# B&R Automation Studio project NAEUL004C00R13L518F00 (part 73)

#### Act_OpsRun2.st
```iecst
(** 2019-04-16 **)
ACTION Act_OpsRun2:

	(*Unloader's Lifter Magazine Layout*)
	(*
		Direction: -->> Left To Right -->>

	                      +----------+
	                      |          |
	                      |          |
	     (Lif=PosCSlt) US3|          |
	               [Mag 3]|          |
	                      |          |
	     (Lif=PosBSlt) US2|          |
	               [Mag 2]|          |
	                      |          |
	     (Lif=PosASlt) US1|          |
	               [Mag 1]|          |
	                      | Unloader |
	                      +----------+

		Note: Program Action Called For Lifter As Shown Above
		      Setup Lifter Program Parameters Accordingly

	For 2 lane magconv
	-eGotoOpsStep, eGotoOpsStep1 will consider lane 1; eGotoOpsStep2,eGotoOpsStep3 consider lane 2
	i. Lifter move position D,E ; Load, Unload pos
	ii. Lifter 2 move position G,H ; Load, Unload pos
	*)

	//===================== third sequence  Lifter 2 ================================================
	IF eGotoOpsStep2 <> eOpsStep2 THEN
		CASE eGotoOpsStep2 OF
			//During unload check ops is standby step
			LiftMagLifterUnload:
				IF eOpsStep = LifMagULStepStandby OR eOpsStep = LifMagULStepMagCmp THEN
					eOpsStep2	:= eGotoOpsStep2;
				END_IF

			LiftMagConvIdle:
				IF eOpsStep2 = LiftMagLifterLoad THEN
					usiMag2Rdy := LifterLoadPos;
					eOpsStep2	:= eGotoOpsStep2;
				ELSIF eOpsStep2 = LiftMagConvOUT THEN
					usiMag2Rdy := LifterNA;
					eOpsStep2	:= eGotoOpsStep2;
				ELSIF eOpsStep2 = LiftMagConvIN THEN
					usiMag2Rdy := LifterMagInProgress;
					eOpsStep2	:= eGotoOpsStep2;
				ELSE
					eOpsStep2	:= eGotoOpsStep2;
				END_IF

			LiftMagConvOUT:
				IF eOpsStep2 = LiftMagLifterUnload THEN
					usiMag2Rdy := LifterUnloadPos;
					eOpsStep2	:= eGotoOpsStep2;
				END_IF

			ELSE
				eOpsStep2	:= eGotoOpsStep2;
		END_CASE
	END_IF

	IF eOpsStep2 = eGotoOpsStep2 THEN
		IF bPaused = FALSE THEN

			CASE eOpsStep2 OF
				LiftMagConvInit:
					sStepTxt1	:= 'Lifter Conveyor 2 Initialization';

					IF bMagSetFullExit2 AND p_bLinkDIOutMagConv2EntSen THEN
						eLifterConv2Act	:= MagConvActExitClpr;
					ELSE
						eLifterConv2Act	:=  MagConvActInitClpStop;
					END_IF

					IF (p_eLifterMagConv2Stat = MagConvActInitClpStop OR p_eLifterMagConv2Stat = MagConvActExitClpr) AND p_eLifterMagConvStatus = Done THEN
						eLifterConv2Act	:= MagConvActIdle;
						eGotoOpsStep2 	:= LifMagULStepInitLif;

					END_IF
					bPaused	:= p_bStop OR p_bStep;

				LifMagULStepInitLif:
					sStepTxt1	:= 'Lifter 2 Initialization';
					IF p_bDIOutShutterCloseRS = TRUE THEN
						eLifter2Act	:= LifterActFullHm;
					END_IF

					IF p_eLifter2Status = Done AND p_eLifter2Stat = LifterActFullHm THEN
						eLifter2Act	:= LifterActIdle;

						eGotoOpsStep2	:= LiftMagConvIdle;

					END_IF
					bPaused	:= p_bStop OR p_bStep;

				LiftMagConvIdle:
					bMagSetFullExit2 := FALSE;
					IF p_bMagConvLanePrep THEN
						IF p_bMagPresentSen2 THEN //limit sensor ON
							//idle,standby
						ELSIF usiMag2Rdy = LifterLoadRdyTrans AND p_bMagPresentSen2 = FALSE THEN //mag2rdy = 2,Lifter inposition (load) and InMagConv ExitSen present
							eGotoOpsStep2 := LiftMagConvIN;
						ELSIF usiMag2Rdy = LifterNA
							AND p_bMagPresentSen2 = FALSE
							AND eOpsStep2 <> LifMagULStepInitLif
							AND p_bOutShutterExtended
							AND p_bLinkDIOutMagConv2EntSen = FALSE
							THEN
							eGotoOpsStep2 :=  LiftMagLifterLoad;
						END_IF

						//Lane 2 prep, magazine2 full
						IF p_bMagConvLanePrep
							AND pa_bMagDis[2] = FALSE
							AND a_bMagAllwMagPresent[2] = TRUE
							AND a_tyMagAllwBffrStat[2].bBffrFull = TRUE
							AND p_bOutShutterExtended
							THEN
							eMagNxtLoad		:= MagNxtLoadInvalid;
							eGotoOpsStep2	:= LiftMagLifterUnload;
						END_IF
					END_IF

					bPaused	:= p_bStop OR p_bStep;

				LiftMagConvIN:
					sStepTxt1	:= 'Lifter 2 Conveyor Entering';
					eLifterConv2Act	:=  MagConvActEntClpStop;

					IF p_eLifterMagConv2Stat = MagConvActEntClpStop AND p_eLifterMagConv2Status = Done THEN
						eLifterConv2Act	:=  MagConvActIdle;
						bLocalMag2InPos := TRUE;
						eGotoOpsStep2 := LiftMagConvIdle;
					END_IF
					bPaused	:= p_bStop OR p_bStep;

				LiftMagConvOUT:
					IF usiMag2Rdy = LifterUnloadRdyTrans THEN //Out mag allow and in position (unload)
						sStepTxt1	:= 'Lifter 2 Conveyor Exiting';
						eLifterConv2Act	:=  MagConvActExitClpr;
						bMagSetFullExit2 := TRUE;
					END_IF

					IF p_eLifterMagConv2Stat = MagConvActExitClpr AND p_eLifterMagConv2Status = Done THEN
						eLifterConv2Act	:=  MagConvActIdle;
						eGotoOpsStep2 := LiftMagConvIdle;
						bMagSetFullExit2 := FALSE;
					END_IF
					bPaused	:= p_bStop OR p_bStep;

				LiftMagLifterLoad:
					sStepTxt1	:= 'Move To Loading Position';
					IF eOpsStep2 <> LifMagULStepInitLif AND bLift2Move = FALSE THEN //AND eOpsStep2 <> LifMagULStepLifMov THEN
						eLifter2Act := LifterActGoGPos; //G,H,; load ,unload
					END_IF

					IF (p_eLifter2Status = Done AND p_eLifter2Stat = LifterActGoGPos)THEN
						eLifter2Act := LifterActIdle;
						eGotoOpsStep2 := LiftMagConvIdle;
					END_IF
					bPaused	:= p_bStop OR p_bStep;

				LiftMagLifterUnload:
					sStepTxt1	:= 'Move To Unload Position';
					IF eOpsStep2 <> LifMagULStepInitLif  AND bLift2Move = FALSE
						AND p_eLifter2Stat <> LifterActGoBSltPos THEN//AND eOpsStep2 <> LifMagULStepLifMov  THEN
						eMagNxtLoad		:= MagNxtLoadInvalid;
						eLifter2Act 	:= LifterActGoHPos; //G,H,; load ,unload
					END_IF

					IF (p_eLifter2Status = Done AND p_eLifter2Stat = LifterActGoHPos)THEN
						eLifter2Act := LifterActIdle;
						eGotoOpsStep2	:= LiftMagConvOUT;
					END_IF
					bPaused	:= p_bStop OR p_bStep;

				LifMagULStepStandby:

			END_CASE
		END_IF
	END_IF
END_ACTION
```

#### Act_OpsInfo.st
```iecst
ACTION Act_OpsInfo:

	//Reset
	udiStatus1	:= 0;
	udiStatus2  := 0;
	//Magazine Not Present
	a_bMagAllwMagPresent[1]	:= p_bMagPresentSen1;
	a_bMagAllwMagPresent[2]	:= p_bMagPresentSen2;
	a_bMagAllwMagPresent[3]	:= p_bMagPresentSen3;

	FOR udi := 1 TO 3 DO
		IF pa_bMagDis[udi] = FALSE AND a_bMagAllwMagPresent[udi] = TRUE THEN
			EXIT;
		END_IF
	END_FOR

	IF udi = 4 THEN
		IF eOpsStep > LifMagULStepInitLif THEN
			udiStatus1	:= 10000;
		END_IF
	END_IF

	//Magazine Is Full
	a_tyMagAllwBffrStat[1]	:= p_tyBufferStat1;
	a_tyMagAllwBffrStat[2]	:= p_tyBufferStat2;
	a_tyMagAllwBffrStat[3]	:= p_tyBufferStat3;

	//Insert Good / Bad Magazine
	IF p_bConvInitDone = TRUE AND p_bConvHvBrd = TRUE THEN

		FOR udi := 1 TO 3 DO
			IF pa_bMagDis[udi] = FALSE AND pa_bMagRej[udi] = TRUE THEN
				EXIT;
			END_IF
		END_FOR

		IF udi < 4 THEN
			//Reject Mode
			IF p_bConvGdBrd = TRUE THEN
				//Good Board Exist
				FOR udi1 := 1 TO 3 DO
					IF pa_bMagDis[udi1] = FALSE AND a_bMagAllwMagPresent[udi1] = TRUE AND pa_bMagRej[udi1] = FALSE THEN
						EXIT;
					END_IF
				END_FOR

				IF udi1 = 4 THEN
					udiStatus1	:= 10004;
				END_IF

			ELSE
				//Bad Board Exist
				FOR udi1 := 1 TO 3 DO
					IF pa_bMagDis[udi1] = FALSE AND a_bMagAllwMagPresent[udi1] = TRUE AND pa_bMagRej[udi1] = TRUE THEN
						EXIT;
					END_IF
				END_FOR

				IF udi1 = 4 THEN
					udiStatus1	:= 10005;
				END_IF

			END_IF

		ELSE
			//Non-Reject Mode
			FOR udi1 := 1 TO 3 DO
				IF pa_bMagDis[udi1] = FALSE AND a_bMagAllwMagPresent[udi1] = TRUE THEN
					EXIT;
				END_IF
			END_FOR

			IF udi1 = 4 THEN
				udiStatus1	:= 10004;
			END_IF

		END_IF

	END_IF

	IF pa_bMagDis[1] = FALSE
		AND pa_bMagDis[2] = FALSE
		AND pa_bMagDis[3] = FALSE
		AND a_bMagAllwMagPresent[1] = TRUE
		AND a_bMagAllwMagPresent[2] = TRUE
		AND a_bMagAllwMagPresent[3] = TRUE
		AND udiStatus1	<> 10008
		THEN

		IF a_tyMagAllwBffrStat[1].bBffrFull
			AND a_tyMagAllwBffrStat[2].bBffrFull
			AND a_tyMagAllwBffrStat[3].bBffrFull
			THEN
			udiStatus1	:= 10008;
		END_IF
	END_IF

	IF pa_bMagDis[1] = FALSE
		AND pa_bMagDis[2] = FALSE
		AND pa_bMagDis[3] = TRUE
		AND a_bMagAllwMagPresent[1] = TRUE
		AND a_bMagAllwMagPresent[2] = TRUE
		AND udiStatus1	<> 10006
		AND udiStatus1	<> 10008
		THEN

		IF (p_tyBufferStat1.diTtlGdBrd + p_tyBufferStat1.diTtlBadBrd
			+ p_tyBufferStat2.diTtlGdBrd + p_tyBufferStat2.diTtlBadBrd >=
			p_tyBufferStat1.diTtlBrdCap + p_tyBufferStat2.diTtlBrdCap - 1)

			THEN
			udiStatus1	:= 10006;

		END_IF
	END_IF

	IF pa_bMagDis[1] = FALSE
			AND pa_bMagDis[2] = FALSE
			AND pa_bMagDis[3] = FALSE
			AND a_bMagAllwMagPresent[1] = TRUE
			AND a_bMagAllwMagPresent[2] = TRUE
			AND a_bMagAllwMagPresent[3] = TRUE
			AND udiStatus1	<> 10007
			AND udiStatus1	<> 10008
			THEN

			IF (p_tyBufferStat1.diTtlGdBrd + p_tyBufferStat1.diTtlBadBrd
			+ p_tyBufferStat2.diTtlGdBrd + p_tyBufferStat2.diTtlBadBrd
			+ p_tyBufferStat3.diTtlGdBrd + p_tyBufferStat3.diTtlBadBrd>=
			p_tyBufferStat1.diTtlBrdCap
			+ p_tyBufferStat2.diTtlBrdCap
			+ p_tyBufferStat3.diTtlBrdCap - 1)

				THEN
				udiStatus1	:= 10007;

			END_IF
	END_IF

	FOR udi := 1 TO 3 DO
		IF pa_bMagDis[udi] = FALSE AND a_bMagAllwMagPresent[udi] = TRUE AND a_tyMagAllwBffrStat[udi].bBffrFull = TRUE THEN
				udiStatus1	:= 10001 + (udi - 1);

			EXIT;
		END_IF
	END_FOR

END_ACTION
```

#### Act_OpsRst.st - Do Not Change!!!
```iecst
(** 2019-03-25 **)
ACTION Act_OpsRst:

	udiStatus1	:= 0;

	eLifterAct		:= LifterActIdle;
	eLifter2Act		:= LifterActIdle;
	eLifterConvAct		:= MagConvActIdle;
	eLifterConv2Act		:= MagConvActIdle;
	eBufferAct1		:= BufferActIdle;
	eBufferAct2		:= BufferActIdle;
	eBufferAct3		:= BufferActIdle;
	eUSSMEMAAct1	:= SMEMAActIdle;
	eUSSMEMAAct2	:= SMEMAActIdle;
	eUSSMEMAAct3	:= SMEMAActIdle;

	usiMag1Rdy 	:= LifterNA;
	usiMag2Rdy	:= LifterNA;
END_ACTION
```

### OpsPosAllwGo.typ - not listed in the package file held
```iecst
(*2018-12-11*)
(**)
(**)
(**)

TYPE
	ePosUSAllwGoStep :
		(
		ePosUSAllwGoStepNA,
		ePosUSAllwGoStepInit,
		ePosUSAllwGoStepStdBy,
		ePosUSAllwGoUSCheck
		);
	ePosDSAllwGoStep :
		(
		ePosDSAllwGoStepNA,
		ePosDSAllwGoStepInit,
		ePosDSAllwGoStepStdBy,
		ePosDSAllwGoDSCheck
		);
END_TYPE
```

### OpsPosAllwGo.var - not listed in the package file held
```iecst
VAR
	p_OpsUSPosAllwGoStep : UDINT;
	p_OpsDSPosAllwGoStep : UDINT;
	p_OpsDSPosAllwGo : UDINT;
	p_OpsUSPosAllwGo : UDINT;
END_VAR
```

### OpsInMagConv.typ - Do Not Change!!!
```iecst
(*2018-12-11*)
(**)
(*Sequence*)

TYPE
	eInMagConvStep :
		(
		InMagConvStepNA,
		InMagConvStepInit,
		InMagConvStepChk,
		InMagConvStepOpsEntMag,
		InMagConvStepOpsExtChkMagSize,
		InMagConvStepOpsExtMag,
		InMagConvStepOpsEntToMid
		);
END_TYPE
```

### OpsInMagConv.var - Change By Project
```iecst
(*2019-03-25*)
(**)
(*Action & State & Status*)
(**)
(*Alarm*)
VAR
	p_OpsInMagConvAlmData : UDINT;
END_VAR
(**)
(*Output*)
VAR
	p_OpsInMagConvAct : UDINT;
	p_OpsInMagConv2Act : UDINT;
	p_OpsInMagConvStepTxt : UDINT;
	p_OpsInMagConvStepTxt1 : UDINT;
	p_OpsInMagConvPaused : UDINT;
END_VAR
(**)
VAR
	p_OpsInMagConvStepEntMag : UDINT;
	p_OpsInMagConvStepEntToMid : UDINT;
	p_OpsInMagConvStepExtMag : UDINT;
	p_OpsInMagConvUSSOTAct : UDINT;
	p_OpsInMagConv2USSOTAct : UDINT;
	p_OpsInMagConv2StepEntMag : UDINT;
	p_OpsInMagConv2StepEntToMid : UDINT;
	p_OpsInMagConv2StepExtMag : UDINT;
END_VAR
```

### Program Logical/Operations/MultiMag_InOutMagazineConv/OpsInMagConv (IEC) - 1.00.0 - 

#### InputRef.var
```iecst
(*2019-04-16*)
(**)
(*General*)
VAR
	p_udiRstErr : REFERENCE TO UDINT;
	p_bEn : REFERENCE TO BOOL;
	p_bDis : REFERENCE TO BOOL;
	p_bRun : REFERENCE TO BOOL;
	p_bStop : REFERENCE TO BOOL;
	p_bStep : REFERENCE TO BOOL;
END_VAR
(**)
(*Configuration*)
VAR
	p_eInMagConvStat : REFERENCE TO eMagConvAction;
	p_eInMagConvStatus : REFERENCE TO eFBStatus;
	p_eInMagConv2Stat : REFERENCE TO eMagConvAction;
	p_eInMagConv2Status : REFERENCE TO eFBStatus;
END_VAR
(**)
VAR
	p_bStepOpsEntMag : REFERENCE TO BOOL;
	p_bStepOpsEntMidMag : REFERENCE TO BOOL;
	p_bStepOpsExtMag : REFERENCE TO BOOL;
	p_bStepOpsEntMag2 : REFERENCE TO BOOL;
	p_bStepOpsEntMidMag2 : REFERENCE TO BOOL;
	p_bStepOpsExtMag2 : REFERENCE TO BOOL;
END_VAR
(**)
VAR
	p_bMagSelMiniMag : REFERENCE TO BOOL;
END_VAR
(**)
VAR
	p_bInMagConvExtSen : REFERENCE TO BOOL;
	p_bMagHeightChkSen : REFERENCE TO BOOL;
	p_eLiftMagConvStatus : REFERENCE TO eFBStatus;
	p_eLiftMagConv2Status : REFERENCE TO eFBStatus;
END_VAR
(**)
(*AGV SOT*)
VAR
	p_eAGVMagStat : REFERENCE TO eAGVMagAction;
	p_eAGVMagStatus : REFERENCE TO eFBStatus;
	p_bAGVMagMcRunRdy : REFERENCE TO BOOL;
	p_eUSSOTStat : REFERENCE TO eSOTAction;
	p_eUSSOTStatus : REFERENCE TO eFBStatus;
	p_eUSSOTStat2 : REFERENCE TO eSOTAction;
	p_eUSSOTStatus2 : REFERENCE TO eFBStatus;
	p_bUSSOTTransporting : REFERENCE TO BOOL;
	p_bUSSOTTransporting2 : REFERENCE TO BOOL;
	p_bUSSOTConvStart : REFERENCE TO BOOL;
	p_bUSSOTConvStop : REFERENCE TO BOOL;
	p_bUSSOTUSRdy : REFERENCE TO BOOL;
END_VAR
(**)
VAR
	p_sProgNm : REFERENCE TO STRING[15];
	p_bNtSettingsLoadDone : REFERENCE TO BOOL;
	p_bCurtainSensorStat : REFERENCE TO BOOL;
END_VAR
```

#### InputRef_Link.var
```iecst
(*2018-12-11*)
(**)
(*External Data*)
VAR
	p_bLinkOpsLifMagULInitDone1 : REFERENCE TO BOOL;
	p_bLinkOpsLifMagULInitDone2 : REFERENCE TO BOOL;
	p_diLinkLifterActualPos : REFERENCE TO DINT;
	p_diLinkLifter2ActualPos : REFERENCE TO DINT;
	p_diLinkLifterTopPos : REFERENCE TO DINT;
	p_diLinkLifterTopPos2 : REFERENCE TO DINT;
	bLifterTopPos : BOOL;
	bLifterTopPos2 : BOOL;
	p_bLinkExtStprExtended : REFERENCE TO BOOL;
	p_bLinkExtStprRetracted : REFERENCE TO BOOL;
	p_bLinkExtStpr2Retracted : REFERENCE TO BOOL;
	p_bLinkInMagConvEntSen : REFERENCE TO BOOL;
	p_bLinkInMagConvExtSen : REFERENCE TO BOOL;
	p_bLinkInMagConvMidSen : REFERENCE TO BOOL;
	p_bLinkInMagConv2EntSen : REFERENCE TO BOOL;
	p_bLinkInMagConv2ExtSen : REFERENCE TO BOOL;
	p_bLinkInMagConv2MidSen : REFERENCE TO BOOL;
	p_bLinkUIMagRun : REFERENCE TO BOOL;
	p_bLinkOpsLifterMagStepEntMag : REFERENCE TO BOOL;
	p_bLinkOpsLifterMagStepExtMag : REFERENCE TO BOOL;
	p_bLinkOpsLifterMagStepEntMag2 : REFERENCE TO BOOL;
	p_bLinkOpsLifterMagStepExtMag2 : REFERENCE TO BOOL;
	p_eLinkMcParamMagExMode : REFERENCE TO eMcMagExchangeMode;
END_VAR
```

#### Local.var
```iecst
(*2019-04-16*)
(**)
(*Local Action, State & Status*)
VAR
	eStatus : eFBStatus := Idle;
	udiStatus : UDINT := 0;
	udiStatus1 : UDINT := 0;
END_VAR
(**)
(*Local Alarm*)
VAR
	tyAlmData : tyAlmDat;
	a_tyAlmText : ARRAY[10000..10099] OF tyAlmTxt := [(sAlmText:='Invalid Magazine Size.'),(sAlmText:='Top Magazine Conveyor Full.'),98((0))];
END_VAR
(**)
(*Local Output*)
VAR
	sStepTxt : STRING[80];
	sStepTxt1 : STRING[80];
	bPaused : BOOL;
	bStepEnterMag : BOOL := FALSE;
	bStepEntToMid : BOOL := FALSE;
	bStepExitMag : BOOL := FALSE;
	bStepEnterMag2 : BOOL := FALSE;
	bStepEntToMid2 : BOOL := FALSE;
	bStepExitMag2 : BOOL := FALSE;
END_VAR
(**)
VAR
	eInMagConvAct : eMagConvAction;
	eInMagConv2Act : eMagConvAction;
END_VAR
(**)
(*Local Input*)
VAR
	udiRstErr : UDINT := 0;
	bEn : BOOL := TRUE;
	bDis : BOOL := FALSE;
	bRun : BOOL;
	bStop : BOOL;
	bStep : BOOL;
END_VAR
(**)
VAR
	eInMagConvStat : eMagConvAction;
	eInMagConvStatus : eFBStatus;
	eInMagConv2Stat : eMagConvAction;
	eInMagConv2Status : eFBStatus;
	eUSSOTAct : eSOTAction;
	eUSSOTAct2 : eSOTAction;
END_VAR
(**)
VAR
	bStepOpsEntMag : BOOL := FALSE;
	bStepOpsEntMidMag : BOOL := FALSE;
	bStepOpsExtMag : BOOL := FALSE;
	bStepOpsEntMag2 : BOOL := FALSE;
	bStepOpsEntMidMag2 : BOOL := FALSE;
	bStepOpsExtMag2 : BOOL := FALSE;
END_VAR
(**)
VAR
	bMagSelMiniMag : BOOL := FALSE;
END_VAR
(**)
VAR
	bInMagConvExtSen : BOOL;
	bMagHeightChkSen : BOOL;
	bCurtainSensorStat : BOOL;
END_VAR
(**)
VAR
	sProgNm : STRING[15] := 'OpsInMagConv';
	bNtSettingsLoadDone : BOOL := TRUE;
END_VAR
(**)
(*Local*)
VAR
	bRstErr : BOOL;
	udiRstErrOld : UDINT;
	bInitialDone : BOOL;
	bInitDone : BOOL;
	eOpsStep : eInMagConvStep := InMagConvStepNA;
	eGotoStep : eInMagConvStep := InMagConvStepInit;
	eOpsStep1 : eInMagConvStep := InMagConvStepNA;
	eGotoStep1 : eInMagConvStep := InMagConvStepInit;
	bMnlLoad : BOOL;
	bMnlLoad2 : BOOL;
	bLiftConvMagExist : BOOL;
	bLiftConvMagExist2 : BOOL;
	bMagManEx : BOOL;
	bMagAutoEx : BOOL;
	udiModuleNum : UDINT := 6111;
END_VAR
```

#### Act_Alarm.st
```iecst
(** 2019-03-25 **)
ACTION Act_Alarm:

	//Error
	IF EDGEPOS(eStatus = Error) THEN

		tyAlmData.sProgNm		:= p_sProgNm;
		tyAlmData.udiCode		:= udiStatus;
		tyAlmData.eSeverity		:= AlmSeverityError;
		tyAlmData.udiRunTime	:= tyAlmData.udiRunTime + 1;
		tyAlmData.bAlm			:= TRUE;
		tyAlmData.udiModuleNum  := udiModuleNum;
		g_sOpsInMagConvProgNm		:= p_sProgNm;

		//Get Error Message
		IF tyAlmData.udiCode < 10000 OR tyAlmData.udiCode > 10099 THEN
			tyAlmData.sAlmMsg	:= 'Unknown';
			tyAlmData.sRcyMsg	:= 'Unknown';
		ELSE
			tyAlmData.sAlmMsg	:= a_tyAlmText[tyAlmData.udiCode].sAlmText;
			tyAlmData.sRcyMsg	:= a_tyAlmText[tyAlmData.udiCode].sRcyText;
		END_IF

	ELSIF bRstErr AND (tyAlmData.udiCode <> 0) THEN

		tyAlmData.udiCode		:= 0;
		tyAlmData.eSeverity		:= AlmSeverityNA;
		tyAlmData.sAlmMsg		:= '';
		tyAlmData.sRcyMsg		:= '';
		tyAlmData.bAlm			:= FALSE;
	END_IF

END_ACTION
```

#### Act_AlarmInfo.st
```iecst
(** 2019-01-14 **)
ACTION Act_AlarmInfo:

	//Info
	tyAlmData.sProgNm		:= p_sProgNm;
	tyAlmData.udiCode		:= udiStatus1;
	tyAlmData.eSeverity		:= AlmSeverityInfo;
	tyAlmData.udiRunTime	:= tyAlmData.udiRunTime + 1;

	//Get Info Message
	IF tyAlmData.udiCode < 10000 OR tyAlmData.udiCode > 10099 THEN
		tyAlmData.sAlmMsg	:= 'Unknown';
		tyAlmData.sRcyMsg	:= 'Unknown';
	ELSE
		tyAlmData.sAlmMsg	:= a_tyAlmText[tyAlmData.udiCode].sAlmText;
		tyAlmData.sRcyMsg	:= a_tyAlmText[tyAlmData.udiCode].sRcyText;
	END_IF

END_ACTION
```

#### Act_Background.st
```iecst
(** 2019-04-16 **)
ACTION Act_Background:

	//Reset bPaused
	IF EDGENEG(p_bStop OR p_bStep) THEN
		bPaused	:= FALSE;
	END_IF

	IF eStatus <> Error AND p_bRun = TRUE THEN
		IF (p_bEn = TRUE) AND (p_bDis = FALSE) THEN
			Act_OpsRun;
			Act_OpsInMagInfo;
		ELSE
			bPaused	:= p_bStop OR p_bStep;
		END_IF

		IF EDGEPOS(p_bEn = FALSE OR p_bDis = TRUE) THEN
			Act_OpsRst;
		END_IF

	ELSIF eStatus <> Error THEN
		sStepTxt	:= 'Stop';
		sStepTxt1	:= 'Stop';
	ELSE
		sStepTxt	:= 'Error';
		sStepTxt1	:= 'Error';
	END_IF

	//Reset
	IF EDGENEG(p_bRun) OR EDGEPOS(eStatus = Error) THEN
		Act_OpsInitial;
		Act_OpsRst;
	END_IF

	//Reset Error
	IF (eStatus = Error) AND bRstErr THEN
		eStatus		:= Idle;
		udiStatus	:= 0;
	END_IF

END_ACTION
```

#### Act_InitGlobal.st
```iecst
(** 2019-04-16 **)
ACTION Act_InitGlobal:

	(* Always Change If Project Change *)

	//Pass Data To Link
	p_bLinkOpsLifMagULInitDone1 ACCESS p_OpsLifMagULStepInitDone1;
	p_bLinkOpsLifMagULInitDone2 ACCESS p_OpsLifMagULStepInitDone2;
	p_diLinkLifterActualPos ACCESS p_LifterBtmActualPos;
	p_diLinkLifter2ActualPos ACCESS p_Lifter2ActualPos;
	p_diLinkLifterTopPos ACCESS p_McParamLifterTopPos;
	p_diLinkLifterTopPos2 ACCESS p_McParamLifterTopPos2;
	p_bLinkExtStprExtended ACCESS p_PneuNoSenTopExtStprExtended;
	p_bLinkExtStprRetracted ACCESS p_PneuNoSenTopExtStprRetracted;
	p_bLinkExtStpr2Retracted ACCESS p_PneuNoSenTopExtStpr2Retracted;
	p_bLinkInMagConvEntSen ACCESS p_DIInMagConvEntSen;
	p_bLinkInMagConvExtSen ACCESS p_DIInMagConvExtSen;
	p_bLinkInMagConvMidSen ACCESS p_DIInMagConvMidSen;
	p_bLinkInMagConv2EntSen ACCESS p_DIInMagConv2EntSen;
	p_bLinkInMagConv2ExtSen ACCESS p_DIInMagConv2ExtSen;
	p_bLinkInMagConv2MidSen ACCESS p_DIInMagConv2MidSen;
	//	p_bLinkUIMagRun ACCESS p_UIMagRun;
	p_bLinkOpsLifterMagStepEntMag ACCESS p_OpsLifMagULStepEntMag1;
	p_bLinkOpsLifterMagStepExtMag ACCESS p_OpsLifMagULStepExtMag1;
	p_bLinkOpsLifterMagStepEntMag2 ACCESS p_OpsLifMagULStepEntMag2;
	p_bLinkOpsLifterMagStepExtMag2 ACCESS p_OpsLifMagULStepExtMag2;
	p_eLinkMcParamMagExMode ACCESS p_McParamMagExMode;

	//Pass Data To Internal Use
	p_udiRstErr ACCESS p_RstErrReset;
//	p_bEn ACCESS p_OpsLifMagULStepInitDone1;
	p_bRun ACCESS p_OpsRun;
	p_bStop ACCESS p_OpsStop;
	p_bStep ACCESS p_OpsStep;

	p_eInMagConvStat ACCESS p_InMagConvStat;
	p_eInMagConvStatus ACCESS p_InMagConvStatus;
	p_eInMagConv2Stat ACCESS p_InMagConv2Stat;
	p_eInMagConv2Status ACCESS p_InMagConv2Status;

	p_bInMagConvExtSen ACCESS p_DIInMagConvExtSen;
//	p_bMagHeightChkSen ACCESS p_DIMagHeightChkSen;

	p_eLiftMagConvStatus ACCESS p_LifterMagConvStatus;
	p_eLiftMagConv2Status ACCESS p_LifterMagConv2Status;

	//AGV
	p_eAGVMagStat ACCESS p_AGVMag1Stat;
	p_eAGVMagStatus ACCESS p_AGVMag1Status;
	p_bAGVMagMcRunRdy ACCESS p_AGVMag1McRunRdy;
	//USSOT
	p_eUSSOTStat ACCESS p_USSOT1Stat;
	p_eUSSOTStatus ACCESS p_USSOT1Status;
	p_bUSSOTTransporting ACCESS p_USSOT1Transporting;
	p_bUSSOTConvStart ACCESS p_USSOT1ConvStart;
	p_bUSSOTConvStop ACCESS p_USSOT1ConvStop;
	p_bUSSOTUSRdy ACCESS p_USSOT1USRdy;
	p_eUSSOTStat2 ACCESS p_USSOT2Stat;
	p_eUSSOTStatus2 ACCESS p_USSOT2Status;
	p_bUSSOTTransporting2 ACCESS p_USSOT2Transporting;

	//	p_bMagSelMiniMag ACCESS p_MagRcpCurrRcpMiniMag;

//	p_sProgNm ACCESS p_NtParamOpsULDInMagProgNm;
	p_bNtSettingsLoadDone ACCESS p_StartupNtSettingsLoadDone;
//	p_bCurtainSensorStat ACCESS p_CurtainSensorStat;

	(* Always Change If Project Change *)

END_ACTION
```

#### Act_InitLocal.st
```iecst
(** 2019-04-16 **)
ACTION Act_InitLocal:

	//Input Reference Link To Local Variable
	p_udiRstErr ACCESS ADR(udiRstErr);
	p_bEn ACCESS ADR(bEn);
	p_bDis ACCESS ADR(bDis);
	p_bRun ACCESS ADR(bRun);
	p_bStop ACCESS ADR(bStop);
	p_bStep ACCESS ADR(bStep);

	p_eInMagConvStat ACCESS ADR(eInMagConvStat);
	p_eInMagConvStatus ACCESS ADR(eInMagConvStatus);
	p_eInMagConv2Stat ACCESS ADR(eInMagConv2Stat);
	p_eInMagConv2Status ACCESS ADR(eInMagConv2Status);

	p_bStepOpsEntMag ACCESS ADR(bStepOpsEntMag);
	p_bStepOpsEntMidMag ACCESS ADR(bStepOpsEntMidMag);
	p_bStepOpsExtMag ACCESS ADR(bStepOpsExtMag);
	p_bStepOpsEntMag2 ACCESS ADR(bStepOpsEntMag2);
	p_bStepOpsEntMidMag2 ACCESS ADR(bStepOpsEntMidMag2);
	p_bStepOpsExtMag2 ACCESS ADR(bStepOpsExtMag2);

	p_bMagSelMiniMag ACCESS ADR(bMagSelMiniMag);

	p_bMagHeightChkSen ACCESS ADR(bMagHeightChkSen);
	p_bInMagConvExtSen ACCESS ADR(bInMagConvExtSen);
	p_bCurtainSensorStat ACCESS ADR(bCurtainSensorStat);

	p_sProgNm ACCESS ADR(sProgNm);
	p_bNtSettingsLoadDone ACCESS ADR(bNtSettingsLoadDone);

END_ACTION
```

#### Act_Link.st
```iecst
(** 2018-12-11 **)
ACTION Act_Link:

	bLifterTopPos		:= (ABS(p_diLinkLifterActualPos - p_diLinkLifterTopPos))<500;
	bLifterTopPos2		:= (ABS(p_diLinkLifter2ActualPos - p_diLinkLifterTopPos2))<500;

//	p_bStepOpsEntMag	:= p_bLinkOpsLifMagULInitDone1 = TRUE AND (p_bLinkUIMagRun = TRUE OR (p_bLinkInMagConvExtSen = FALSE AND p_bLinkInMagConvMidSen = TRUE));
	p_bStepOpsEntMag	:= p_bLinkInMagConvExtSen = FALSE AND p_bLinkInMagConvMidSen = TRUE;
	p_bStepOpsExtMag	:= p_bLinkOpsLifMagULInitDone1 = TRUE AND bLifterTopPos = TRUE AND p_bLinkExtStprRetracted = TRUE AND p_bLinkInMagConvExtSen = TRUE AND p_bLinkOpsLifterMagStepEntMag = TRUE;
	p_bStepOpsEntMidMag	:= p_bLinkInMagConvEntSen AND p_bLinkInMagConvMidSen = FALSE;

	p_bStepOpsEntMag2	:= p_bLinkInMagConv2ExtSen = FALSE AND p_bLinkInMagConv2MidSen = TRUE;
	p_bStepOpsExtMag2	:= p_bLinkOpsLifMagULInitDone2 = TRUE AND bLifterTopPos2 = TRUE AND p_bLinkExtStpr2Retracted = TRUE AND p_bLinkInMagConv2ExtSen = TRUE AND p_bLinkOpsLifterMagStepEntMag2 = TRUE;
	p_bStepOpsEntMidMag2:= p_bLinkInMagConv2EntSen AND p_bLinkInMagConv2MidSen = FALSE;

	//LiftConv Out magazine
	IF p_bLinkOpsLifterMagStepExtMag THEN
		bLiftConvMagExist := FALSE;
	END_IF
	IF p_bLinkOpsLifterMagStepExtMag2 THEN
		bLiftConvMagExist2 := FALSE;
	END_IF

	//Mag Exchange Mode
	CASE p_eLinkMcParamMagExMode OF
		McSetMagXcAutoManMode:
			bMagManEx := TRUE;
			bMagAutoEx := TRUE;

		McSetMagXcAutoMode:
			bMagManEx := FALSE;
			bMagAutoEx := TRUE;

		McSetMagXcManMode:
			bMagManEx := TRUE;
			bMagAutoEx := FALSE;

	END_CASE
END_ACTION
```

#### Init.st
```iecst
(** 2019-03-25 **)
PROGRAM _INIT

	(* Always Change If Project Change *)

	//Pass Address To Global Address For External Use
	//Action, State & Status

	//Alarm
	p_OpsInMagConvAlmData		:= ADR(tyAlmData);

	//Output
	p_OpsInMagConvAct			:= ADR(eInMagConvAct);
	p_OpsInMagConv2Act			:= ADR(eInMagConv2Act);
	p_OpsInMagConvUSSOTAct		:= ADR(eUSSOTAct);
	p_OpsInMagConv2USSOTAct		:= ADR(eUSSOTAct2);
	p_OpsInMagConvStepTxt		:= ADR(sStepTxt);
	p_OpsInMagConvStepTxt1		:= ADR(sStepTxt1);
	p_OpsInMagConvPaused		:= ADR(bPaused);

	p_OpsInMagConvStepEntMag	:= ADR(bStepEnterMag);
	p_OpsInMagConvStepEntToMid	:= ADR(bStepEntToMid);
	p_OpsInMagConvStepExtMag	:= ADR(bStepExitMag);

	p_OpsInMagConv2StepEntMag	:= ADR(bStepEnterMag2);
	p_OpsInMagConv2StepEntToMid	:= ADR(bStepEntToMid2);
	p_OpsInMagConv2StepExtMag	:= ADR(bStepExitMag2);

	(* Always Change If Project Change *)

END_PROGRAM
```

#### Act_OpsInitial.st - Do Not Change!!!
```iecst
(** 2019-01-16 **)
ACTION Act_OpsInitial:

	eGotoStep	:= InMagConvStepInit;
	eOpsStep	:= InMagConvStepNA;
	eGotoStep1	:= InMagConvStepInit;
	eOpsStep1	:= InMagConvStepNA;

	bStepEnterMag	:= FALSE;
	bStepEntToMid 	:= FALSE;
	bStepExitMag	:= FALSE;
	bStepEnterMag2	:= FALSE;
	bStepEntToMid2	:= FALSE;
	bStepExitMag2	:= FALSE;

END_ACTION
```

#### Act_OpsInMagInfo.st
```iecst
(** 2019-04-16 **)
ACTION Act_OpsInMagInfo:

	IF p_bLinkInMagConvMidSen = TRUE AND p_bLinkInMagConvExtSen = TRUE AND p_bCurtainSensorStat = TRUE THEN
		udiStatus1		:= 10001;//Top magazine conveyor full.
	ELSE
		udiStatus1		:= 0;
	END_IF

END_ACTION
```

#### Act_OpsRun.st
```iecst
(** 2019-04-16 **)
ACTION Act_OpsRun:

	IF eGotoStep <> eOpsStep THEN

		CASE eGotoStep OF

			ELSE
				eOpsStep	:= eGotoStep;

		END_CASE

	END_IF

	IF eGotoStep = eOpsStep THEN

		IF bPaused = FALSE THEN

			CASE eOpsStep OF
				InMagConvStepNA:
					sStepTxt	:= 'NA';

					eGotoStep	:= InMagConvStepInit;

					//					bPaused		:= p_bStop OR p_bStep;

				InMagConvStepInit:
					sStepTxt			:= 'Initializing Magazine Conveyor';
					eInMagConvAct		:= MagConvActInit;

					IF (p_eInMagConvStatus = Done AND p_eInMagConvStat = MagConvActInit)
						THEN
						eInMagConvAct			:= MagConvActIdle;
						eGotoStep			:= InMagConvStepChk;
					END_IF

				InMagConvStepChk:
					sStepTxt	:= 'Checking Input Magazine Conveyor Condition';

					IF bMagAutoEx AND p_bLinkInMagConvMidSen = FALSE THEN
						eUSSOTAct	:= SOTActRun;
					ELSE
						eUSSOTAct	:= SOTActIdle;
					END_IF

					IF p_bStepOpsExtMag = TRUE AND bLiftConvMagExist = FALSE THEN
						eGotoStep	:= InMagConvStepOpsExtMag;
					ELSIF p_bStepOpsEntMag = TRUE THEN
						eGotoStep	:= InMagConvStepOpsEntMag;
					ELSIF p_bUSSOTTransporting= TRUE THEN 		//SOT Comm
						eGotoStep	:= InMagConvStepOpsEntToMid;
					ELSIF p_bStepOpsEntMidMag = TRUE THEN
						bMnlLoad	:= TRUE;
						eGotoStep	:= InMagConvStepOpsEntToMid;
					END_IF

					IF p_bStepOpsExtMag = FALSE AND p_bStepOpsEntMag = FALSE AND p_eLiftMagConvStatus <> Busy THEN
						bPaused		:= p_bStop OR p_bStep;
						IF bPaused THEN
							eUSSOTAct	:= SOTActIdle;
						END_IF
					END_IF

				InMagConvStepOpsEntMag:
					sStepTxt	:= 'Entering Magazine';

					eInMagConvAct		:= MagConvActInit;

					IF p_eInMagConvStatus = Done AND p_eInMagConvStat = MagConvActInit THEN
						eInMagConvAct	:= MagConvActIdle;
						eGotoStep		:= InMagConvStepChk;

						bPaused	:= p_bStop OR p_bStep;
					END_IF

				InMagConvStepOpsExtChkMagSize:
					sStepTxt	:= 'Checking Magazine Size';

					IF p_bMagSelMiniMag = TRUE THEN
						IF p_bMagHeightChkSen = TRUE AND p_bInMagConvExtSen = TRUE THEN
							eStatus		:= Error;
							udiStatus	:= 10000;		// Invalid Magazine Size
						ELSE
							eGotoStep	:= InMagConvStepOpsExtMag;
						END_IF
					ELSE
						eGotoStep	:= InMagConvStepOpsExtMag;
					END_IF

				InMagConvStepOpsExtMag:
					sStepTxt	:= 'Exiting Magazine';

					eInMagConvAct		:= MagConvActExit;

					IF p_eInMagConvStatus = Done AND p_eInMagConvStat = MagConvActExit THEN
						bLiftConvMagExist := TRUE;
						eInMagConvAct	:= MagConvActIdle;
						eGotoStep		:= InMagConvStepChk;

						bPaused	:= p_bStop OR p_bStep;
					END_IF

				InMagConvStepOpsEntToMid:
					sStepTxt	:= 'Entering Magazine To Middle';

					eInMagConvAct		:= MagConvActInit;

					IF p_eInMagConvStatus = Done AND p_eInMagConvStat = MagConvActInit AND
						(bMnlLoad OR (p_eUSSOTStatus = Done AND p_eUSSOTStat = SOTActRun)) THEN
						bMnlLoad		:= FALSE;
						eInMagConvAct	:= MagConvActIdle;
						eUSSOTAct		:= SOTActIdle;
						eGotoStep		:= InMagConvStepChk;

						bPaused	:= p_bStop OR p_bStep;
					END_IF

			END_CASE

		END_IF

	ELSE
		bPaused	:= p_bStop OR p_bStep;

	END_IF

	Act_OpsRun2;

	//Operation Step Status
	bStepEnterMag		:= eOpsStep = InMagConvStepOpsEntMag;
	bStepEntToMid		:= eOpsStep = InMagConvStepOpsEntToMid;
	bStepExitMag		:= eOpsStep = InMagConvStepOpsExtMag;

END_ACTION
```

#### Act_OpsRun2.st
```iecst
(** 2019-04-16 **)
ACTION Act_OpsRun2:
	//InMagConv Lane2
	//**********************second sequence - InMag2 ********************************************************
	IF eGotoStep1 <> eOpsStep1 THEN

		CASE eGotoStep1 OF

			ELSE
				eOpsStep1	:= eGotoStep1;

		END_CASE

	END_IF

	IF eGotoStep1 = eOpsStep1 THEN

		IF bPaused = FALSE THEN

			CASE eOpsStep1 OF
				InMagConvStepNA:
					sStepTxt1	:= 'NA';

					eGotoStep1	:= InMagConvStepInit;

//					bPaused		:= p_bStop OR p_bStep;

				InMagConvStepInit:
					sStepTxt1			:= 'Initializing Magazine Conveyor';
					eInMagConv2Act		:= MagConvActInit;

					IF (p_eInMagConv2Status = Done AND p_eInMagConv2Stat = MagConvActInit)
						THEN
						eInMagConv2Act			:= MagConvActIdle;
						eGotoStep1				:= InMagConvStepChk;
					END_IF

				InMagConvStepChk:
					sStepTxt1	:= 'Checking Input Magazine Conveyor Condition';

					IF bMagAutoEx AND p_bLinkInMagConv2MidSen = FALSE THEN
						eUSSOTAct2	:= SOTActRun;
					ELSE
						eUSSOTAct2	:= SOTActIdle;
					END_IF

					IF p_bStepOpsExtMag2 = TRUE AND bLiftConvMagExist2 = FALSE THEN
						eGotoStep1	:= InMagConvStepOpsExtMag;
					ELSIF p_bStepOpsEntMag2 = TRUE THEN
						eGotoStep1	:= InMagConvStepOpsEntMag;
					ELSIF  p_bUSSOTTransporting2= TRUE THEN		//SOT Comm
						eGotoStep1	:= InMagConvStepOpsEntToMid;
					ELSIF p_bStepOpsEntMidMag2 = TRUE THEN
						bMnlLoad2	:= TRUE;
						eGotoStep1	:= InMagConvStepOpsEntToMid;
					END_IF

					IF p_bStepOpsExtMag2 = FALSE AND p_bStepOpsEntMag2 = FALSE AND p_eLiftMagConv2Status <> Busy THEN
						bPaused		:= p_bStop OR p_bStep;
						IF bPaused THEN
							eUSSOTAct2	:= SOTActIdle;
						END_IF
					END_IF

				InMagConvStepOpsEntMag:
					sStepTxt1	:= 'Entering Magazine';

					eInMagConv2Act		:= MagConvActInit;

					IF p_eInMagConv2Status = Done AND p_eInMagConv2Stat = MagConvActInit THEN
						eInMagConv2Act	:= MagConvActIdle;
						eGotoStep1		:= InMagConvStepChk;

						bPaused	:= p_bStop OR p_bStep;
					END_IF

				InMagConvStepOpsExtChkMagSize:
					sStepTxt1	:= 'Checking Magazine Size';

					IF p_bMagSelMiniMag = TRUE THEN
						IF p_bMagHeightChkSen = TRUE AND p_bInMagConvExtSen = TRUE THEN
							eStatus		:= Error;
							udiStatus	:= 10000;		// Invalid Magazine Size
						ELSE
							eGotoStep1	:= InMagConvStepOpsExtMag;
						END_IF
					ELSE
						eGotoStep1	:= InMagConvStepOpsExtMag;
					END_IF

				InMagConvStepOpsExtMag:
					sStepTxt1	:= 'Exiting Magazine';

					eInMagConv2Act		:= MagConvActExit;

					IF p_eInMagConv2Status = Done AND p_eInMagConv2Stat = MagConvActExit THEN
						bLiftConvMagExist2 := TRUE;
						eInMagConv2Act	:= MagConvActIdle;
						eGotoStep1		:= InMagConvStepChk;

						bPaused	:= p_bStop OR p_bStep;
					END_IF

				InMagConvStepOpsEntToMid:
					sStepTxt1	:= 'Entering Magazine To Middle';

					eInMagConv2Act		:= MagConvActInit;

					IF p_eInMagConv2Status = Done AND p_eInMagConv2Stat = MagConvActInit AND
						(bMnlLoad2 OR  (p_eUSSOTStatus2 = Done AND p_eUSSOTStat2 = SOTActRun)) THEN
						bMnlLoad2		:= FALSE;
						eInMagConv2Act	:= MagConvActIdle;
						eUSSOTAct2		:= SOTActIdle;
						eGotoStep1		:= InMagConvStepChk;

						bPaused	:= p_bStop OR p_bStep;
					END_IF

			END_CASE

		END_IF

	ELSE
		bPaused	:= p_bStop OR p_bStep;
	END_IF

	//Operation Step Status
	bStepEnterMag2		:= eOpsStep1 = InMagConvStepOpsEntMag;
	bStepEntToMid2		:= eOpsStep1 = InMagConvStepOpsEntToMid;
	bStepExitMag2		:= eOpsStep1 = InMagConvStepOpsExtMag;

END_ACTION
```

#### Act_OpsRst.st - Do Not Change!!!
```iecst
(** 2019-03-25 **)
ACTION Act_OpsRst:

	eInMagConvAct	:= MagConvActIdle;
	eInMagConv2Act	:= MagConvActIdle;
	eUSSOTAct	:= SOTActIdle;
	eUSSOTAct2	:= SOTActIdle;
	bMnlLoad	:= FALSE;
	bMnlLoad2	:= FALSE;

END_ACTION
```

### OpsOutMagConv.typ - Do Not Change!!!
```iecst
(*2018-12-11*)
(**)
(*Sequence*)

TYPE
	eOutMagConvStep :
		(
		OutMagConvStepNA,
		OutMagConvStepInit,
		OutMagConvStepChk,
		OutMagConvStepEntMag,
		OutMagConvStepEntToMid,
		OutMagConvStepExitMag,
		OutMagConvStepWaitForRmvMag
		);
END_TYPE
```

### OpsOutMagConv.var - Change By Project
```iecst
(*2019-03-25*)
(**)
(*Action & State & Status*)
(**)
(*Alarm*)
VAR
	p_OpsOutMagConvAlmData : UDINT;
END_VAR
(**)
(*Output*)
VAR
	p_OpsOutMagConvAct : UDINT;
	p_OpsOutMagConv2Act : UDINT;
	p_OpsOutMagConvDSSOTAct : UDINT;
	p_OpsOutMagConv2DSSOTAct : UDINT;
	p_OpsOutMagConvStepTxt : UDINT;
	p_OpsOutMagConvStepTxt1 : UDINT;
	p_OpsOutMagConvPaused : UDINT;
END_VAR
(**)
VAR
	p_OpsOutMagConvStepInitDone : UDINT;
	p_OpsOutMagConvStepEntMag : UDINT;
	p_OpsOutMagConvStepEntMidMag : UDINT;
	p_OpsOutMagConvStepExtMag : UDINT;
	p_OpsOutMagConvStepWaitToRmvMag : UDINT;
	p_OpsOutMagConv2StepInitDone : UDINT;
	p_OpsOutMagConv2StepEntMag : UDINT;
	p_OpsOutMagConv2StepEntMidMag : UDINT;
	p_OpsOutMagConv2StepExtMag : UDINT;
	p_OpsOutMagConv2StepWaitToRmvMag : UDINT;
END_VAR
```

### Program Logical/Operations/MultiMag_InOutMagazineConv/OpsOutMagConv (IEC) - 1.00.0 - 

#### InputRef.var
```iecst
(*2019-04-16*)
(**)
(*General*)
VAR
	p_udiRstErr : REFERENCE TO UDINT;
	p_bEn : REFERENCE TO BOOL;
	p_bDis : REFERENCE TO BOOL;
	p_bRun : REFERENCE TO BOOL;
	p_bStop : REFERENCE TO BOOL;
	p_bStep : REFERENCE TO BOOL;
END_VAR
(**)
(*Configuration*)
VAR
	p_eOutMagConvStat : REFERENCE TO eMagConvAction;
	p_eOutMagConvStatus : REFERENCE TO eFBStatus;
	p_eOutMagConv2Stat : REFERENCE TO eMagConvAction;
	p_eOutMagConv2Status : REFERENCE TO eFBStatus;
END_VAR
(**)
VAR
	p_bStepEntMag : REFERENCE TO BOOL;
	p_bStepEntMag2 : REFERENCE TO BOOL;
	p_bEntSen : REFERENCE TO BOOL;
	p_bMidSen : REFERENCE TO BOOL;
	p_bExtSen : REFERENCE TO BOOL;
	p_bEntSen2 : REFERENCE TO BOOL;
	p_bMidSen2 : REFERENCE TO BOOL;
	p_bExtSen2 : REFERENCE TO BOOL;
	p_bExitSig : REFERENCE TO BOOL;
	p_bExitSig2 : REFERENCE TO BOOL;
	p_bOpsMnlUnloadMag : REFERENCE TO BOOL;
	p_bOpsMnlUnloadMag2 : REFERENCE TO BOOL;
END_VAR
(**)
(*AGV SOT*)
VAR
	p_eAGVMagStat : REFERENCE TO eAGVMagAction;
	p_eAGVMagStatus : REFERENCE TO eFBStatus;
	p_bAGVMagMcRunRdy : REFERENCE TO BOOL;
	p_eDSSOTStat : REFERENCE TO eSOTAction;
	p_eDSSOTStatus : REFERENCE TO eFBStatus;
	p_eDSSOTStat2 : REFERENCE TO eSOTAction;
	p_eDSSOTStatus2 : REFERENCE TO eFBStatus;
	p_bDSSOTTransporting : REFERENCE TO BOOL;
	p_bDSSOTTransporting2 : REFERENCE TO BOOL;
	p_bDSSOTConvStart : REFERENCE TO BOOL;
	p_bDSSOTConvStop : REFERENCE TO BOOL;
END_VAR
(**)
VAR
	p_sProgNm : REFERENCE TO STRING[15];
	p_bNtSettingsLoadDone : REFERENCE TO BOOL;
END_VAR
```

#### InputRef_Link.var
```iecst
(*2018-12-11*)
(**)
(*External Data*)
VAR
	p_bLinkOpsLifMagULInitDone1 : REFERENCE TO BOOL;
	p_bLinkOpsLifMagULInitDone2 : REFERENCE TO BOOL;
	p_diLinkLifterActualPos : REFERENCE TO DINT;
	p_diLinkLifterBtmPos : REFERENCE TO DINT;
	p_diLinkLifter2ActualPos : REFERENCE TO DINT;
	p_diLinkLifterBtmPos2 : REFERENCE TO DINT;
	bLifterBtmPos : BOOL;
	bLifterBtmPos2 : BOOL;
	p_tyLinkBffrStat : REFERENCE TO tyBffrStat;
	p_tyLinkBffr2Stat : REFERENCE TO tyBffrStat;
	p_bLinkLifterLmtSW : REFERENCE TO BOOL;
	p_bLinkLifter2LmtSW : REFERENCE TO BOOL;
	p_bLinkLiftExitMag : REFERENCE TO BOOL;
	p_bLinkLiftExitMag2 : REFERENCE TO BOOL;
	p_tyLinkDISetting : REFERENCE TO tyDigitalInputSettings;
	p_eLinkMcParamMagExMode : REFERENCE TO eMcMagExchangeMode;
END_VAR
```

#### Local.var
```iecst
(*2019-04-16*)
(**)
(*Local Action, State & Status*)
VAR
	eStatus : eFBStatus := Idle;
	udiStatus : UDINT := 0;
END_VAR
(**)
(*Local Alarm*)
VAR
	tyAlmData : tyAlmDat;
	a_tyAlmText : ARRAY[10000..10099] OF tyAlmTxt;
END_VAR
(**)
(*Local Output*)
VAR
	sStepTxt : STRING[80];
	sStepTxt1 : STRING[80];
	bPaused : BOOL;
	bStepInitDone : BOOL := FALSE;
	bStepEnterMag : BOOL := FALSE;
	bStepEnterMidMag : BOOL := FALSE;
	bStepExitMag : BOOL := FALSE;
	bStepWaitMagToRmvMnl : BOOL := FALSE;
	bStepInitDone2 : BOOL := FALSE;
	bStepEnterMag2 : BOOL := FALSE;
	bStepEnterMidMag2 : BOOL := FALSE;
	bStepExitMag2 : BOOL := FALSE;
	bStepWaitMagToRmvMnl2 : BOOL := FALSE;
END_VAR
(**)
VAR
	eOutMagConvAct : eMagConvAction;
	eOutMagConv2Act : eMagConvAction;
	eDSSOTAct : eSOTAction;
	eDSSOTAct2 : eSOTAction;
END_VAR
(**)
(*Local Input*)
VAR
	udiRstErr : UDINT := 0;
	bEn : BOOL := TRUE;
	bDis : BOOL := FALSE;
	bRun : BOOL;
	bStop : BOOL;
	bStep : BOOL;
END_VAR
(**)
VAR
	eOutMagConvStat : eMagConvAction;
	eOutMagConvStatus : eFBStatus;
	eOutMagConv2Stat : eMagConvAction;
	eOutMagConv2Status : eFBStatus;
END_VAR
(* *)
VAR
	bStepEntMag : BOOL := FALSE;
	bStepEntMag2 : BOOL := FALSE;
	bEntSen : BOOL := FALSE;
	bMidSen : BOOL := FALSE;
	bExtSen : BOOL := FALSE;
	bEntSen2 : BOOL := FALSE;
	bMidSen2 : BOOL := FALSE;
	bExtSen2 : BOOL := FALSE;
	bExitSig : BOOL := FALSE;
	bExitSig2 : BOOL := FALSE;
	bOpsMnlUnloadMag : BOOL := FALSE;
	fbMagToRmv : TON := (IN:=TRUE,PT:=T#1s);
	fbMagToRmv2 : TON := (IN:=TRUE,PT:=T#1s);
END_VAR
(**)
VAR
	sProgNm : STRING[15] := 'OpsAW';
	bNtSettingsLoadDone : BOOL := TRUE;
END_VAR
(**)
(*Local*)
VAR
	bRstErr : BOOL;
	udiRstErrOld : UDINT;
	bInitialDone : BOOL;
	bInitDone : BOOL;
	eOpsStep : eOutMagConvStep := OutMagConvStepNA;
	eGotoStep : eOutMagConvStep := OutMagConvStepInit;
	eOpsStep1 : eOutMagConvStep := OutMagConvStepNA;
	eGotoStep1 : eOutMagConvStep := OutMagConvStepInit;
	bMagManEx : BOOL;
	bMagAutoEx : BOOL;
	udiModuleNum : UDINT := 6131;
END_VAR
```

#### Act_Alarm.st
```iecst
(** 2019-03-25 **)
ACTION Act_Alarm:

	//Error
	IF EDGEPOS(eStatus = Error) THEN

		tyAlmData.sProgNm		:= p_sProgNm;
		tyAlmData.udiCode		:= udiStatus;
		tyAlmData.eSeverity		:= AlmSeverityError;
		tyAlmData.udiRunTime	:= tyAlmData.udiRunTime + 1;
		tyAlmData.bAlm			:= TRUE;
		tyAlmData.udiModuleNum  := udiModuleNum;
		g_sOpsOutMagConvProgNm		:= p_sProgNm;
		//Get Error Message
		IF tyAlmData.udiCode < 10000 OR tyAlmData.udiCode > 10099 THEN
			tyAlmData.sAlmMsg	:= 'Unknown';
			tyAlmData.sRcyMsg	:= 'Unknown';
		ELSE
			tyAlmData.sAlmMsg	:= a_tyAlmText[tyAlmData.udiCode].sAlmText;
			tyAlmData.sRcyMsg	:= a_tyAlmText[tyAlmData.udiCode].sRcyText;
		END_IF

	ELSIF bRstErr AND (tyAlmData.udiCode <> 0) THEN

		tyAlmData.udiCode		:= 0;
		tyAlmData.eSeverity		:= AlmSeverityNA;
		tyAlmData.sAlmMsg		:= '';
		tyAlmData.sRcyMsg		:= '';
		tyAlmData.bAlm			:= FALSE;
	END_IF

END_ACTION
```

#### Act_Background.st
```iecst
(** 2019-04-16 **)
ACTION Act_Background:

	//Reset bPaused
	IF EDGENEG(p_bStop OR p_bStep) THEN
		bPaused	:= FALSE;
	END_IF

	IF eStatus <> Error AND p_bRun = TRUE THEN
		IF (p_bEn = TRUE) AND (p_bDis = FALSE) THEN
			Act_OpsRun;
		ELSE
			bPaused	:= p_bStop OR p_bStep;
		END_IF

		IF EDGEPOS(p_bEn = FALSE OR p_bDis = TRUE) THEN
			Act_OpsRst;
		END_IF

	ELSIF eStatus <> Error THEN
		sStepTxt	:= 'Stop';
		sStepTxt1	:= 'Stop';
	ELSE
		sStepTxt	:= 'Error';
		sStepTxt1	:= 'Error';
	END_IF

	//Reset
	IF EDGENEG(p_bRun) OR EDGEPOS(eStatus = Error) THEN
		Act_OpsInitial;
		Act_OpsRst;
	END_IF

	//Reset Error
	IF (eStatus = Error) AND bRstErr THEN
		eStatus		:= Idle;
		udiStatus	:= 0;
	END_IF

END_ACTION
```

#### Act_InitGlobal.st
```iecst
(** 2019-04-16 **)
ACTION Act_InitGlobal:

	(* Always Change If Project Change *)

	//Pass Data To Link
	p_bLinkOpsLifMagULInitDone1 ACCESS p_OpsLifMagULStepInitDone1;
	p_bLinkOpsLifMagULInitDone2 ACCESS p_OpsLifMagULStepInitDone2;
	p_diLinkLifterActualPos ACCESS p_LifterBtmActualPos;
	p_diLinkLifterBtmPos ACCESS p_McParamLifterBtmPos;
	p_diLinkLifter2ActualPos ACCESS p_Lifter2ActualPos;
	p_diLinkLifterBtmPos2 ACCESS p_McParamLifterBtmPos2;
	p_tyLinkBffrStat ACCESS p_Buffer1BffrStat;
	p_tyLinkBffr2Stat ACCESS p_Buffer2BffrStat;
	p_bLinkLifterLmtSW ACCESS p_DILifterLmtSW;
	p_bLinkLifter2LmtSW ACCESS p_DILifter2LmtSW;
	p_bLinkLiftExitMag	ACCESS p_OpsLifMagULStepExtMag1;
	p_bLinkLiftExitMag2	ACCESS p_OpsLifMagULStepExtMag2;
	p_tyLinkDISetting ACCESS p_NtParamDISettings;
	p_eLinkMcParamMagExMode ACCESS p_McParamMagExMode;

	//Pass Data To Internal Use
	p_udiRstErr ACCESS p_RstErrReset;
//	p_bEn ACCESS p_OpsInitULDStepInitDone;
	p_bRun ACCESS p_OpsRun;
	p_bStop ACCESS p_OpsStop;
	p_bStep ACCESS p_OpsStep;

	p_eOutMagConvStat ACCESS p_OutMagConvStat;
	p_eOutMagConvStatus ACCESS p_OutMagConvStatus;
	p_eOutMagConv2Stat ACCESS p_OutMagConv2Stat;
	p_eOutMagConv2Status ACCESS p_OutMagConv2Status;

	p_bEntSen ACCESS p_DIOutMagConvEntSen;
	p_bMidSen ACCESS p_DIOutMagConvMidSen;
	p_bExtSen ACCESS p_DIOutMagConvExtSen;
	p_bEntSen2 ACCESS p_DIOutMagConv2EntSen;
	p_bMidSen2 ACCESS p_DIOutMagConv2MidSen;
	p_bExtSen2 ACCESS p_DIOutMagConv2ExtSen;

	//p_bExitSig ACCESS ADR(bExitSig);

	//AGV
	p_eAGVMagStat ACCESS p_AGVMag1Stat;
	p_eAGVMagStatus ACCESS p_AGVMag1Status;
	p_bAGVMagMcRunRdy ACCESS p_AGVMag1McRunRdy;
	//DSSOT
	p_eDSSOTStat ACCESS p_DSSOT1Stat;
	p_eDSSOTStatus ACCESS p_DSSOT1Status;
	p_eDSSOTStat2 ACCESS p_DSSOT2Stat;
	p_eDSSOTStatus2 ACCESS p_DSSOT2Status;
	p_bDSSOTTransporting ACCESS p_DSSOT1Transporting;
	p_bDSSOTTransporting2 ACCESS p_DSSOT2Transporting;
	p_bDSSOTConvStart ACCESS p_DSSOT1ConvStart;
	p_bDSSOTConvStop ACCESS p_DSSOT1ConvStop;

	p_bOpsMnlUnloadMag ACCESS p_UIOpsMnlUnloadMag;
	p_bOpsMnlUnloadMag2 ACCESS p_UIOpsMnlUnloadMag2;

//	p_sProgNm ACCESS p_NtParamOpsULDOutMagProgNm;
	p_bNtSettingsLoadDone ACCESS p_StartupNtSettingsLoadDone;

	(* Always Change If Project Change *)

END_ACTION
```

#### Act_InitLocal.st
```iecst
(** 2019-04-16 **)
ACTION Act_InitLocal:

	//Output Reference Link To Local Variable
	p_udiRstErr ACCESS ADR(udiRstErr);
	p_bEn ACCESS ADR(bEn);
	p_bDis ACCESS ADR(bDis);
	p_bRun ACCESS ADR(bRun);
	p_bStop ACCESS ADR(bStop);
	p_bStep ACCESS ADR(bStep);

	p_eOutMagConvStat ACCESS ADR(eOutMagConvStat);
	p_eOutMagConvStatus ACCESS ADR(eOutMagConvStatus);
	p_eOutMagConv2Stat ACCESS ADR(eOutMagConv2Stat);
	p_eOutMagConv2Status ACCESS ADR(eOutMagConv2Status);

	p_bStepEntMag ACCESS ADR(bStepEntMag);
	p_bStepEntMag2 ACCESS ADR(bStepEntMag2);
	p_bEntSen ACCESS ADR(bEntSen);
	p_bMidSen ACCESS ADR(bMidSen);
	p_bExtSen ACCESS ADR(bExtSen);
	p_bEntSen2 ACCESS ADR(bEntSen2);
	p_bMidSen2 ACCESS ADR(bMidSen2);
	p_bExtSen2 ACCESS ADR(bExtSen2);
	p_bExitSig ACCESS ADR(bExitSig);
	p_bExitSig2 ACCESS ADR(bExitSig2);
	p_bOpsMnlUnloadMag ACCESS ADR(bOpsMnlUnloadMag);

	p_sProgNm ACCESS ADR(sProgNm);
	p_bNtSettingsLoadDone ACCESS ADR(bNtSettingsLoadDone);

END_ACTION
```

#### Act_Link.st
```iecst
(** 2018-12-11 **)
ACTION Act_Link:

	bLifterBtmPos	:= (ABS(p_diLinkLifterActualPos - p_diLinkLifterBtmPos))<500;
	bLifterBtmPos2	:= (ABS(p_diLinkLifter2ActualPos - p_diLinkLifterBtmPos2))<500;

	p_bStepEntMag	:= p_bLinkOpsLifMagULInitDone1 = TRUE AND bLifterBtmPos = TRUE AND (p_tyLinkBffrStat.bBffrFull = TRUE AND p_bLinkLifterLmtSW = TRUE) AND p_bLinkLiftExitMag;
	p_bStepEntMag2	:= p_bLinkOpsLifMagULInitDone2 = TRUE AND bLifterBtmPos2 = TRUE AND (p_tyLinkBffr2Stat.bBffrFull = TRUE AND p_bLinkLifter2LmtSW = TRUE) AND p_bLinkLiftExitMag2;

	//Mag Exchange Mode
	CASE p_eLinkMcParamMagExMode OF
		McSetMagXcAutoManMode:
			bMagManEx := TRUE;
			bMagAutoEx := TRUE;

		McSetMagXcAutoMode:
			bMagManEx := FALSE;
			bMagAutoEx := TRUE;

		McSetMagXcManMode:
			bMagManEx := TRUE;
			bMagAutoEx := FALSE;
	END_CASE

END_ACTION
```

#### Init.st
```iecst
(** 2019-03-25 **)
PROGRAM _INIT

	(* Always Change If Project Change *)

	//Pass Address To Global Address For External Use
	//Action, State & Status

	//Alarm
	p_OpsOutMagConvAlmData		:= ADR(tyAlmData);

	//Output
	p_OpsOutMagConvAct			:= ADR(eOutMagConvAct);
	p_OpsOutMagConv2Act			:= ADR(eOutMagConv2Act);
	p_OpsOutMagConvDSSOTAct		:= ADR(eDSSOTAct);
	p_OpsOutMagConv2DSSOTAct	:= ADR(eDSSOTAct2);
	p_OpsOutMagConvStepTxt		:= ADR(sStepTxt);
	p_OpsOutMagConvStepTxt1		:= ADR(sStepTxt1);
	p_OpsOutMagConvPaused		:= ADR(bPaused);

	p_OpsOutMagConvStepInitDone		:= ADR(bStepInitDone);
	p_OpsOutMagConvStepEntMag		:= ADR(bStepEnterMag);
	p_OpsOutMagConvStepEntMidMag	:= ADR(bStepEnterMidMag);
	p_OpsOutMagConvStepExtMag		:= ADR(bStepExitMag);
	p_OpsOutMagConvStepWaitToRmvMag	:= ADR(bStepWaitMagToRmvMnl);

	p_OpsOutMagConv2StepInitDone	:= ADR(bStepInitDone2);
	p_OpsOutMagConv2StepEntMag		:= ADR(bStepEnterMag2);
	p_OpsOutMagConv2StepEntMidMag	:= ADR(bStepEnterMidMag2);
	p_OpsOutMagConv2StepExtMag		:= ADR(bStepExitMag2);
	p_OpsOutMagConv2StepWaitToRmvMag	:= ADR(bStepWaitMagToRmvMnl2);

	(* Always Change If Project Change *)

END_PROGRAM
```

#### Act_OpsInitial.st - Do Not Change!!!
```iecst
(** 2019-01-16 **)
ACTION Act_OpsInitial:

	eGotoStep	:= OutMagConvStepInit;
	eOpsStep	:= OutMagConvStepNA;
	eGotoStep1	:= OutMagConvStepInit;
	eOpsStep1	:= OutMagConvStepNA;

	bStepEnterMag		:= FALSE;
	bStepEnterMidMag 	:= FALSE;
	bStepExitMag		:= FALSE;
	bStepEnterMag2		:= FALSE;
	bStepEnterMidMag2 	:= FALSE;
	bStepExitMag2		:= FALSE;

END_ACTION
```

#### Act_OpsRun.st
```iecst
(** 2019-04-16 **)
ACTION Act_OpsRun:

	IF eGotoStep <> eOpsStep THEN

		CASE eGotoStep OF
			OutMagConvStepEntMag:
				IF bMagAutoEx AND p_bExtSen = FALSE THEN
					eDSSOTAct	:= SOTActIdle;
				END_IF

				IF p_bStepEntMag = TRUE THEN
					eOpsStep	:= eGotoStep;
				ELSIF p_bMidSen AND p_bExtSen = FALSE AND p_eOutMagConvStat = MagConvActIdle THEN
					eOpsStep	:= eGotoStep;
				ELSIF p_bMidSen = FALSE AND p_bExtSen THEN
					eGotoStep	:= OutMagConvStepChk;
				ELSIF p_bEntSen = FALSE AND p_bMidSen AND p_bExtSen THEN
					eGotoStep	:= OutMagConvStepEntToMid;
				END_IF

			OutMagConvStepEntToMid:
				IF bMagAutoEx AND p_bExtSen THEN
					eDSSOTAct	:= SOTActRun;
				ELSE
					eDSSOTAct	:= SOTActIdle;
				END_IF

				IF  p_bExtSen = FALSE THEN
					eGotoStep	:= OutMagConvStepChk;
				ELSIF p_bDSSOTTransporting = TRUE THEN
					eGotoStep	:= OutMagConvStepExitMag;
				ELSIF p_bEntSen AND p_bMidSen = FALSE AND p_bExtSen THEN
					eOpsStep	:= eGotoStep;
				ELSIF p_bStepEntMag = TRUE THEN
					eOpsStep	:= eGotoStep;
				ELSIF p_bOpsMnlUnloadMag AND p_bExtSen THEN
					eGotoStep	:= OutMagConvStepWaitForRmvMag;
				END_IF
			ELSE
				eOpsStep		:= eGotoStep;

		END_CASE

	END_IF

	IF eGotoStep = eOpsStep THEN

		IF bPaused = FALSE THEN

			CASE eOpsStep OF
				OutMagConvStepNA:
					sStepTxt	:= 'Output Magazine Conveyor Standby';

					eGotoStep	:= OutMagConvStepInit;

					bPaused		:= p_bStop OR p_bStep;

				OutMagConvStepInit:
					sStepTxt			:= 'Initializing Magazine Conveyor';
					eOutMagConvAct		:= MagConvActInit;

					IF (p_eOutMagConvStatus = Done AND p_eOutMagConvStat = MagConvActInit)
						THEN
						eOutMagConvAct			:= MagConvActIdle;
						eGotoStep				:= OutMagConvStepChk;
					END_IF

				OutMagConvStepChk:
					sStepTxt	:= 'Magazine Checking';
					IF p_tyLinkDISetting.diOutMagConvExtSen <> 0 AND p_bExtSen = FALSE THEN
						eGotoStep		:= OutMagConvStepEntMag;
					ELSIF p_tyLinkDISetting.diOutMagConvMidSen <> 0 AND p_bMidSen = FALSE THEN
						eGotoStep		:= OutMagConvStepEntToMid;
					ELSIF  p_tyLinkDISetting.diOutMagConvEntSen <> 0 AND p_bEntSen = FALSE AND
						p_tyLinkDISetting.diOutMagConvMidSen = 0 AND
						p_tyLinkDISetting.diOutMagConvMidSen = 0 THEN //when only 1 EntSen
						eGotoStep		:= OutMagConvStepEntMag;
					ELSIF (p_bExitSig OR p_bDSSOTTransporting) AND p_bExtSen THEN
						eGotoStep		:= OutMagConvStepExitMag;
					ELSIF p_bExtSen AND p_bMidSen AND p_bOpsMnlUnloadMag = FALSE THEN
						IF bMagAutoEx AND p_bExtSen THEN
							eDSSOTAct	:= SOTActRun;
						ELSE
							eDSSOTAct	:= SOTActIdle;
						END_IF
					ELSIF p_bOpsMnlUnloadMag AND p_bExtSen THEN
						eGotoStep	:= OutMagConvStepWaitForRmvMag;
					END_IF

					bPaused		:= p_bStop OR p_bStep;

				OutMagConvStepEntMag:
					sStepTxt	:= 'Entering Magazine'; //enter to end (extsen)

					eOutMagConvAct		:= MagConvActEnt;

					IF p_eOutMagConvStatus = Done AND p_eOutMagConvStat = MagConvActEnt THEN
						eOutMagConvAct	:= MagConvActIdle;
						eGotoStep		:= OutMagConvStepChk;

						bPaused	:= p_bStop OR p_bStep;
					END_IF

				OutMagConvStepEntToMid:
					sStepTxt	:= 'Entering To Middle Magazine Conveyor';

					eOutMagConvAct		:= MagConvActEnt;

					IF p_eOutMagConvStatus = Done AND p_eOutMagConvStat = MagConvActEnt THEN
						eOutMagConvAct	:= MagConvActIdle;
						eGotoStep		:= OutMagConvStepChk;

						bPaused	:= p_bStop OR p_bStep;
					END_IF

				OutMagConvStepExitMag:
					sStepTxt	:= 'Exiting Magazine';

					eOutMagConvAct		:= MagConvActExit;

					IF p_eOutMagConvStatus = Done AND p_eOutMagConvStat = MagConvActExit AND
						p_eDSSOTStatus = Done AND p_eDSSOTStat = SOTActRun THEN

						eOutMagConvAct		:= MagConvActIdle;
						eDSSOTAct			:= SOTActIdle;
						eGotoStep			:= OutMagConvStepChk;

						bPaused	:= p_bStop OR p_bStep;
					END_IF

				OutMagConvStepWaitForRmvMag:

					sStepTxt  := 'Waiting Magazine To Remove Manually';

					eDSSOTAct   := SOTActIdle;
					fbMagToRmv(IN:= (p_bExtSen = FALSE));

					IF p_bOpsMnlUnloadMag = FALSE OR fbMagToRmv.Q THEN
						fbMagToRmv (IN:= FALSE);
						eGotoStep		:= OutMagConvStepChk;
					END_IF

					bPaused			:= p_bStop OR p_bStep;
			END_CASE

		END_IF

	ELSE
		bPaused	:= p_bStop OR p_bStep;
	END_IF

	Act_OpsRun2;

	//Operation Step Status
	bStepInitDone		:= eOpsStep > OutMagConvStepInit;
	bStepEnterMag		:= eOpsStep = OutMagConvStepEntMag;
	bStepEnterMidMag	:= eOpsStep	= OutMagConvStepEntToMid;
	bStepExitMag		:= eOpsStep = OutMagConvStepExitMag;
	bStepWaitMagToRmvMnl:= eOpsStep = OutMagConvStepWaitForRmvMag;

END_ACTION
```

#### Act_OpsRun2.st
```iecst
(** 2019-04-16 **)
ACTION Act_OpsRun2:
	//OutMagConv Lane2
	//***************** sequence 2  ****************************************************************
	IF eGotoStep1 <> eOpsStep1 THEN

		CASE eGotoStep1 OF
			OutMagConvStepEntMag:
				IF bMagAutoEx AND p_bExtSen2 = FALSE THEN
					eDSSOTAct2	:= SOTActIdle;
				END_IF

				IF p_bStepEntMag2 = TRUE THEN
					eOpsStep1	:= eGotoStep1;
				ELSIF p_bMidSen2 AND p_bExtSen2 = FALSE AND p_eOutMagConv2Stat = MagConvActIdle THEN
					eOpsStep1	:= eGotoStep1;
				ELSIF p_bMidSen2 = FALSE AND p_bExtSen2 THEN
					eGotoStep1	:= OutMagConvStepChk;
				ELSIF p_bEntSen2 = FALSE AND p_bMidSen2 AND p_bExtSen2 THEN
					eGotoStep1	:= OutMagConvStepEntToMid;
				END_IF

			OutMagConvStepEntToMid:
				IF bMagAutoEx AND p_bExtSen2 THEN
					eDSSOTAct2	:= SOTActRun;
				ELSE
					eDSSOTAct2	:= SOTActIdle;
				END_IF

				IF  p_bExtSen2 = FALSE THEN
					eGotoStep1	:= OutMagConvStepChk;
				ELSIF p_bDSSOTTransporting2 = TRUE THEN
					eGotoStep1	:= OutMagConvStepExitMag;
				ELSIF p_bEntSen2 AND p_bMidSen2 = FALSE AND p_bExtSen2 THEN
					eOpsStep1	:= eGotoStep1;
				ELSIF p_bStepEntMag2 = TRUE THEN
					eOpsStep1	:= eGotoStep1;
				ELSIF p_bOpsMnlUnloadMag2 AND p_bExtSen2 THEN
					eGotoStep1	:= OutMagConvStepWaitForRmvMag;
				END_IF
			ELSE
				eOpsStep1		:= eGotoStep1;

		END_CASE

	END_IF

	IF eGotoStep1 = eOpsStep1 THEN

		IF bPaused = FALSE THEN

			CASE eOpsStep1 OF
				OutMagConvStepNA:
					sStepTxt1	:= 'Output Magazine Conveyor Standby';

					eGotoStep1	:= OutMagConvStepInit;

					bPaused		:= p_bStop OR p_bStep;

				OutMagConvStepInit:
					sStepTxt1			:= 'Initializing Magazine Conveyor';
					eOutMagConv2Act		:= MagConvActInit;

					IF (p_eOutMagConv2Status = Done AND p_eOutMagConv2Stat = MagConvActInit)
						THEN
						eOutMagConv2Act			:= MagConvActIdle;
						eGotoStep1				:= OutMagConvStepChk;
					END_IF

				OutMagConvStepChk:
					sStepTxt1	:= 'Magazine Checking';
					IF p_tyLinkDISetting.diOutMagConv2ExtSen <> 0 AND p_bExtSen2 = FALSE THEN
						eGotoStep1		:= OutMagConvStepEntMag;
					ELSIF p_tyLinkDISetting.diOutMagConv2MidSen <> 0 AND p_bMidSen2 = FALSE THEN
						eGotoStep1		:= OutMagConvStepEntToMid;
					ELSIF  p_tyLinkDISetting.diOutMagConv2EntSen <> 0 AND p_bEntSen2 = FALSE AND
						p_tyLinkDISetting.diOutMagConvMidSen = 0 AND
						p_tyLinkDISetting.diOutMagConvMidSen = 0 THEN //when only 1 EntSen
						eGotoStep1		:= OutMagConvStepEntMag;
					ELSIF (p_bExitSig2 OR p_bDSSOTTransporting2) AND p_bExtSen2 THEN
						eGotoStep1		:= OutMagConvStepExitMag;
					ELSIF p_bExtSen2 AND p_bMidSen2 AND p_bOpsMnlUnloadMag2 = FALSE THEN
						IF bMagAutoEx AND p_bExtSen2 THEN
							eDSSOTAct2	:= SOTActRun;
						ELSE
							eDSSOTAct2	:= SOTActIdle;
						END_IF
					ELSIF p_bOpsMnlUnloadMag2 AND p_bExtSen2 THEN
						eGotoStep1	:= OutMagConvStepWaitForRmvMag;
					END_IF

					bPaused		:= p_bStop OR p_bStep;

				OutMagConvStepEntMag:
					sStepTxt1	:= 'Entering Magazine'; //enter to end (extsen)

					eOutMagConv2Act		:= MagConvActEnt;

					IF p_eOutMagConv2Status = Done AND p_eOutMagConv2Stat = MagConvActEnt THEN
						eOutMagConv2Act	:= MagConvActIdle;
						eGotoStep1		:= OutMagConvStepChk;

						bPaused	:= p_bStop OR p_bStep;
					END_IF

				OutMagConvStepEntToMid:
					sStepTxt1	:= 'Entering To Middle Magazine Conveyor';

					eOutMagConv2Act		:= MagConvActEnt;

					IF p_eOutMagConv2Status = Done AND p_eOutMagConv2Stat = MagConvActEnt THEN
						eOutMagConv2Act	:= MagConvActIdle;
						eGotoStep1		:= OutMagConvStepChk;

						bPaused	:= p_bStop OR p_bStep;
					END_IF

				OutMagConvStepExitMag:
					sStepTxt1	:= 'Exiting Magazine';

					eOutMagConv2Act		:= MagConvActExit;

					IF p_eOutMagConv2Status = Done AND p_eOutMagConv2Stat = MagConvActExit AND
						p_eDSSOTStatus2 = Done AND p_eDSSOTStat2 = SOTActRun THEN

						eOutMagConv2Act		:= MagConvActIdle;
						eDSSOTAct2			:= SOTActIdle;
						eGotoStep1			:= OutMagConvStepChk;

						bPaused	:= p_bStop OR p_bStep;
					END_IF

				OutMagConvStepWaitForRmvMag:

					sStepTxt1  := 'Waiting Magazine To Remove Manually';

					eDSSOTAct2   := SOTActIdle;
					fbMagToRmv2(IN:= (p_bExtSen2 = FALSE));

					IF p_bOpsMnlUnloadMag2 = FALSE OR fbMagToRmv2.Q THEN
						fbMagToRmv2 (IN:= FALSE);
						eGotoStep1		:= OutMagConvStepChk;
					END_IF

					bPaused			:= p_bStop OR p_bStep;
			END_CASE

		END_IF

	ELSE
		bPaused	:= p_bStop OR p_bStep;
	END_IF

	//Operation Step Status
	bStepInitDone2		:= eOpsStep1 	> OutMagConvStepInit;
	bStepEnterMag2		:= eOpsStep1 	= OutMagConvStepEntMag;
	bStepEnterMidMag2	:= eOpsStep1	= OutMagConvStepEntToMid;
	bStepExitMag2		:= eOpsStep1	= OutMagConvStepExitMag;
	bStepWaitMagToRmvMnl2:= eOpsStep1 	= OutMagConvStepWaitForRmvMag;

END_ACTION
```

#### Act_OpsRst.st - Do Not Change!!!
```iecst
(** 2019-03-25 **)
ACTION Act_OpsRst:

	eOutMagConvAct	:= MagConvActIdle;
	eOutMagConv2Act	:= MagConvActIdle;
	eDSSOTAct	:= SOTActIdle;

END_ACTION
```

### OpsMagConvStpr.typ - Do Not Change!!!
```iecst
(*2018-12-11*)
(**)
(*Sequence*)

TYPE
	eMagConvStprRunStep :
		(
		MagConvStprStepNA,
		MagConvStprStepInit,
		MagConvStprStepChkCond,
		MagConvStprStepBtmLiftMagEnt,
		MagConvStprStepBtmLiftMagExit,
		MagConvStprStepTopLiftMagEnt,
		MagConvStprStepTopLiftMagExit,
		MagConvStprStepTopMagConvEnter,
		MagConvStprStepTopMagConvEnterD,
		MagConvStprStepBtmMagConvExit,
		MagConvStprStepDone,
		MagConvStprStepInitDone,
		MagConvStprStepBtmMagExitMnl
		);
END_TYPE
```

### OpsMagConvStpr.var - Change By Project
```iecst
(*2019-03-25*)
(**)
(*Action & State & Status*)
(**)
(*Alarm*)
VAR
	p_OpsMagConvStprAlmData : UDINT;
END_VAR
(**)
(*Output*)
VAR
	p_OpsMagConvStprStepTxt : UDINT;
	p_OpsMagConvStprPaused : UDINT;
	p_OpsMagConvStprBtmEntAct : UDINT;
	p_OpsMagConvStprBtmExitAct : UDINT;
	p_OpsMagConvStprBtmMidAct : UDINT;
	p_OpsMagConvStprTopEntAct : UDINT;
	p_OpsMagConvStprTopExitAct : UDINT;
	p_OpsMagConvStprTopMidAct : UDINT;
END_VAR
```

### Program Logical/Operations/MultiMag_InOutMagazineConv/OpsMagConvStpr (IEC) - 1.00.0 - 

#### Act_Alarm.st
```iecst
(** 2019-03-25 **)
ACTION Act_Alarm:

	//Error
	IF EDGEPOS(eStatus = Error) THEN

		tyAlmData.sProgNm		:= p_sProgNm;
		tyAlmData.udiCode		:= udiStatus;
		tyAlmData.eSeverity		:= AlmSeverityError;
		tyAlmData.udiRunTime	:= tyAlmData.udiRunTime + 1;
		tyAlmData.bAlm			:= TRUE;
		tyAlmData.udiModuleNum  := udiModuleNum;
		g_sOpsMagConvStprProgNm		:= p_sProgNm;
		//Get Error Message
		IF tyAlmData.udiCode < 10000 OR tyAlmData.udiCode > 10099 THEN
			tyAlmData.sAlmMsg	:= 'Unknown';
			tyAlmData.sRcyMsg	:= 'Unknown';
		ELSE
			tyAlmData.sAlmMsg	:= a_tyAlmText[tyAlmData.udiCode].sAlmText;
			tyAlmData.sRcyMsg	:= a_tyAlmText[tyAlmData.udiCode].sRcyText;
		END_IF

	ELSIF bRstErr AND (tyAlmData.udiCode <> 0) THEN

		tyAlmData.udiCode		:= 0;
		tyAlmData.eSeverity		:= AlmSeverityNA;
		tyAlmData.sAlmMsg		:= '';
		tyAlmData.sRcyMsg		:= '';

	END_IF

END_ACTION
```

#### Act_InitGlobal.st
```iecst
(** 2019-04-16 **)
ACTION Act_InitGlobal:

	(* Always Change If Project Change *)

	//Pass Data To Link
	p_bLinkOpsMnlUnloadMag ACCESS p_UIOpsMnlUnloadMag;
	p_bLinkOpsOutMagConvStepWaitRmv ACCESS p_OpsOutMagConvStepWaitToRmvMag;

	//Pass Data To Internal Use
	p_udiRstErr ACCESS p_RstErrReset;
	p_bRun ACCESS p_OpsRun;
	p_bStop ACCESS p_OpsStop;
	p_bStep ACCESS p_OpsStep;
	p_sProgNm ACCESS p_NtParamOpsMagConvStprProgNm;
	p_bNtSettingsLoadDone ACCESS p_StartupNtSettingsLoadDone;

	p_diLinkLiftBtmActualPos ACCESS p_LifterBtmActualPos;
	p_diLinkLiftBtmPos ACCESS p_McParamLifterBtmPos;
	p_diLinkLiftTopPos ACCESS p_McParamLifterTopPos;

	p_eStprBtmMidStat ACCESS p_PneuNoSenBtmMidStprStat;
	p_eStprBtmMidStatus ACCESS p_PneuNoSenBtmMidStprStatus;

	p_eStprBtmExitStat ACCESS p_PneuNoSenBtmExtStprStat;
	p_eStprBtmExitStatus ACCESS p_PneuNoSenBtmExtStprStatus;

	p_eStprTopEntStat ACCESS p_PneuNoSenTopEntStprStat;
	p_eStprTopEntStatus ACCESS p_PneuNoSenTopEntStprStatus;

	p_eStprTopMidStat ACCESS p_PneuNoSenTopMidStprStat;
	p_eStprTopMidStatus ACCESS p_PneuNoSenTopMidStprStatus;
	p_bStprTopMidStprExtended ACCESS p_PneuNoSenTopMidStprExtended;

	p_eStprTopExitStat ACCESS p_PneuNoSenTopExtStprStat;
	p_eStprTopExitStatus ACCESS p_PneuNoSenTopExtStprStatus;
	p_bStprTopExitStprExtended ACCESS p_PneuNoSenTopEntStprExtended;

	p_eInMagConvStatus ACCESS p_InMagConvStatus; 	//In magConv status
	p_eInMagConvStat ACCESS p_InMagConvStat; 	//In magConv status
	p_eOutMagConvStatus ACCESS p_OutMagConvStatus; 	//In magConv status
	p_eLiftMagConvStat ACCESS p_LifterMagConvStat; //LiftConv Status
	p_eLiftMagConvStatus ACCESS p_LifterMagConvStatus;

//	p_bBtmMagConvZ1Sen ACCESS p_DIBtmMagConvZ1Sen;
//	p_bTopMagConvZ1Sen ACCESS p_DITopMagConvZ1Sen;
	p_bBtmMagConvZ1Sen ACCESS p_DIOutMagConvEntSen;
	p_bTopMagConvZ1Sen ACCESS p_DIInMagConvExtSen;

	p_bBtmMagConvMidSen ACCESS p_DIOutMagConvMidSen; //LtoR view
	p_bTopMagConvMidSen ACCESS p_DIInMagConvMidSen;

	p_bBtmMagConvEndSen ACCESS p_DIOutMagConvExtSen; //LtoR view
	p_bTopMagConvEndSen ACCESS p_DIInMagConvEntSen;

	p_bMagPresentSen ACCESS p_DILifterLmtSW;

	p_bEnterSig ACCESS p_OpsInMagConvStepEntToMid;
	p_bExitSig ACCESS p_OpsOutMagConvStepExtMag;

	(* Always Change If Project Change *)

END_ACTION
```

#### Act_Link.st
```iecst
(** 2018-12-11 **)
ACTION Act_Link:

	IF (ABS(p_diLinkLiftBtmActualPos - p_diLinkLiftBtmPos))<500 THEN

		p_bLiftBtmPos	:= TRUE;

	ELSE
		p_bLiftBtmPos	:= FALSE;

	END_IF

	IF (ABS(p_diLinkLiftBtmActualPos - p_diLinkLiftTopPos))<500 THEN

		p_bLiftTopPos	:= TRUE;

	ELSE
		p_bLiftTopPos	:= FALSE;

	END_IF

	p_bBtmEntToLift		:= p_bMagPresentSen = FALSE AND p_bBtmMagConvZ1Sen AND ((p_eLiftMagConvStat = MagConvActEntStopClp (*OR p_eLiftMagConvStat = MagConvActInitStopClp*)) AND p_eLiftMagConvStatus = Busy) AND p_bLiftBtmPos;

	p_bTopExitFromLift	:= (p_eLiftMagConvStat = MagConvActExitClpr AND p_eLiftMagConvStatus = Busy) AND p_bLiftTopPos;

	p_bBtmExitFromLift	:=  (p_eLiftMagConvStat = MagConvActExitClpr AND p_eLiftMagConvStatus = Busy) AND p_bLiftBtmPos;

	p_bTopEntToLift		:= p_bMagPresentSen = FALSE AND p_bTopMagConvZ1Sen
							AND ((p_eLiftMagConvStat = MagConvActEntClpStop)
							AND p_eLiftMagConvStatus = Busy)
							AND p_bLiftTopPos;

	p_bTopEntFromMagConv := p_bEnterSig;// AND p_bTopMagConvEndSen;
	p_bBtmExitFromMagConv := p_bExitSig AND p_bBtmMagConvEndSen;
	p_bBtmExitMnl		 := p_bLinkOpsMnlUnloadMag AND p_bLinkOpsOutMagConvStepWaitRmv AND p_bBtmMagConvEndSen;

END_ACTION
```

#### Init.st
```iecst
(** 2019-03-25 **)
PROGRAM _INIT

	(* Always Change If Project Change *)

	//Pass Address To Global Address For External Use
	//Action, State & Status

	//Alarm
	p_OpsMagConvStprAlmData	:= ADR(tyAlmData);

	//Output
	p_OpsMagConvStprStepTxt		:= ADR(sStepTxt);
	p_OpsMagConvStprPaused		:= ADR(bPaused);
	p_OpsMagConvStprBtmEntAct	:= ADR(eStprBtmEntAct);
	p_OpsMagConvStprBtmExitAct	:= ADR(eStprBtmExitAct);
	p_OpsMagConvStprBtmMidAct   := ADR(eStprBtmMidAct);
	p_OpsMagConvStprTopEntAct	:= ADR(eStprTopEntAct);
	p_OpsMagConvStprTopExitAct	:= ADR(eStprTopExitAct);
	p_OpsMagConvStprTopMidAct	:= ADR(eStprTopMidAct);

	(* Always Change If Project Change *)

END_PROGRAM
```

#### Program Logical/Operations/MultiMag_InOutMagazineConv/OpsMagConvStpr/Sequence

##### Act_OpsRst.st
```iecst
(** 2019-03-25 **)
ACTION Act_OpsRst:

	eStprBtmExitAct	:= PneuActIdle;
	eStprBtmMidAct	:= PneuActIdle;
	eStprTopExitAct := PneuActIdle;
	eStprTopMidAct	:= PneuActIdle;

END_ACTION
```

### OpsMagConvStpr2.var - Change By Project
```iecst
(*2019-03-25*)
(**)
(*Action & State & Status*)
(**)
(*Alarm*)
VAR
	p_OpsMagConv2StprAlmData : UDINT;
END_VAR
(**)
(*Output*)
VAR
	p_OpsMagConv2StprStepTxt : UDINT;
	p_OpsMagConv2StprPaused : UDINT;
	p_OpsMagConv2StprBtmEntAct : UDINT;
	p_OpsMagConv2StprBtmExitAct : UDINT;
	p_OpsMagConv2StprBtmMidAct : UDINT;
	p_OpsMagConv2StprTopEntAct : UDINT;
	p_OpsMagConv2StprTopExitAct : UDINT;
	p_OpsMagConv2StprTopMidAct : UDINT;
END_VAR
```

### Program Logical/Operations/MultiMag_InOutMagazineConv/OpsMagConvStpr2 (IEC) - 1.00.0 - 

#### InputRef.var
```iecst
(*2019-04-16*)
(**)
(*General*)
VAR
	p_udiRstErr : REFERENCE TO UDINT;
	p_bEn : REFERENCE TO BOOL;
	p_bDis : REFERENCE TO BOOL;
	p_bRun : REFERENCE TO BOOL;
	p_bStop : REFERENCE TO BOOL;
	p_bStep : REFERENCE TO BOOL;
END_VAR
(**)
VAR
	p_bBtmEntToLift : REFERENCE TO BOOL;
	p_bBtmExitFromLift : REFERENCE TO BOOL;
	p_bTopEntToLift : REFERENCE TO BOOL;
	p_bTopExitFromLift : REFERENCE TO BOOL;
	p_bTopEntFromMagConv : REFERENCE TO BOOL;
	p_bBtmExitFromMagConv : REFERENCE TO BOOL;
	p_bBtmExitMnl : REFERENCE TO BOOL;
END_VAR
(**)
VAR
	p_eStprTopEntStat : REFERENCE TO ePneuAction;
	p_eStprTopEntStatus : REFERENCE TO eFBStatus;
END_VAR
(**)
VAR
	p_eStprBtmMidStat : REFERENCE TO ePneuAction;
	p_eStprBtmMidStatus : REFERENCE TO eFBStatus;
	p_eStprTopMidStat : REFERENCE TO ePneuAction;
	p_eStprTopMidStatus : REFERENCE TO eFBStatus;
	p_bStprTopMidStprExtended : REFERENCE TO BOOL;
END_VAR
(**)
VAR
	p_eStprBtmExitStat : REFERENCE TO ePneuAction;
	p_eStprBtmExitStatus : REFERENCE TO eFBStatus;
	p_eStprTopExitStat : REFERENCE TO ePneuAction;
	p_eStprTopExitStatus : REFERENCE TO eFBStatus;
	p_bStprTopExitStprExtended : REFERENCE TO BOOL;
END_VAR
(**)
VAR
	p_eLiftMagConvAct : REFERENCE TO eMagConvAction;
	p_eInMagConvStat : REFERENCE TO eMagConvAction;
	p_eInMagConvStatus : REFERENCE TO eFBStatus;
	p_eOutMagConvStatus : REFERENCE TO eFBStatus;
	p_eLiftMagConvStat : REFERENCE TO eMagConvAction;
	p_eLiftMagConvStatus : REFERENCE TO eFBStatus;
	p_bBtmMagConvZ1Sen : REFERENCE TO BOOL;
	p_bTopMagConvZ1Sen : REFERENCE TO BOOL;
	p_bTopMagConvMidSen : REFERENCE TO BOOL;
	p_bBtmMagConvMidSen : REFERENCE TO BOOL;
	p_bBtmMagConvEndSen : REFERENCE TO BOOL;
	p_bTopMagConvEndSen : REFERENCE TO BOOL;
	p_bMagPresentSen : REFERENCE TO BOOL;
END_VAR
(**)
VAR
	p_bLiftBtmPos : REFERENCE TO BOOL;
	p_bLiftTopPos : REFERENCE TO BOOL;
END_VAR
(**)
VAR
	p_bEnterSig : REFERENCE TO BOOL;
	p_bExitSig : REFERENCE TO BOOL;
END_VAR
(**)
VAR
	p_sProgNm : REFERENCE TO STRING[15];
	p_bNtSettingsLoadDone : REFERENCE TO BOOL;
END_VAR
```

#### InputRef_Link.var
```iecst
(*2018-12-11*)
(**)
VAR
	p_diLinkLiftBtmActualPos : REFERENCE TO DINT;
	p_diLinkLiftBtmPos : REFERENCE TO DINT;
	p_diLinkLiftTopPos : REFERENCE TO DINT;
	p_usiLinkProdRcpMcMode : REFERENCE TO USINT;
END_VAR
(**)
VAR
	p_bLinkOpsMnlUnloadMag : REFERENCE TO BOOL;
	p_bLinkOpsOutMagConvStepWaitRmv : REFERENCE TO BOOL;
END_VAR
```

#### Local.var
```iecst
(*2019-04-16*)
(**)
(*Local Action, State & Status*)
VAR
	eStatus : eFBStatus := Idle;
	udiStatus : UDINT := 0;
END_VAR
(**)
(*Local Alarm*)
VAR
	tyAlmData : tyAlmDat;
	a_tyAlmText : ARRAY[10000..10099] OF tyAlmTxt;
END_VAR
(**)
(*Local Output*)
VAR
	sStepTxt : STRING[80];
	bPaused : BOOL;
	eStprBtmEntAct : ePneuAction;
	eStprBtmMidAct : ePneuAction;
	eStprBtmExitAct : ePneuAction;
	eStprTopEntAct : ePneuAction;
	eStprTopMidAct : ePneuAction;
	eStprTopExitAct : ePneuAction;
	eLiftMagConvAct : ePneuAction;
END_VAR
(**)
(*Local Input*)
VAR
	udiRstErr : UDINT := 0;
	bEn : BOOL := TRUE;
	bDis : BOOL := FALSE;
	bRun : BOOL;
	bStop : BOOL;
	bStep : BOOL;
	eStprBtmMidStat : ePneuAction;
	eStprBtmMidStatus : eFBStatus;
	eStprBtmExitStatus : eFBStatus;
	eStprBtmExitStat : ePneuAction;
	eStprTopEntStat : ePneuAction;
	eStprTopEntStatus : eFBStatus;
	eStprTopMidStat : ePneuAction;
	eStprTopMidStatus : eFBStatus;
	eStprTopExitStat : ePneuAction;
	eStprTopExitStatus : eFBStatus;
	bLiftBtmPos : BOOL := FALSE;
	bLiftTopPos : BOOL;
	bBtmMagConvZ1Sen : BOOL;
	bTopMagConvZ1Sen : BOOL;
	bTopMagConvMidSen : BOOL;
	bBtmMagConvMidSen : BOOL;
	bBtmMagConvEndSen : BOOL;
	bTopMagConvEndSen : BOOL;
	bMagPresentSen : BOOL;
	sProgNm : STRING[15] := 'Ops1';
	bNtSettingsLoadDone : BOOL := TRUE;
	bBtmEntToLift : BOOL;
	bBtmExitFromLift : BOOL;
	bTopEntToLift : BOOL;
	bTopExitFromLift : BOOL;
	bTopEntFromMagConv : BOOL;
	bBtmExitFromMagConv : BOOL;
	bBtmExitMnl : BOOL;
	bEnterSig : BOOL;
	bExitSig : BOOL;
END_VAR
(**)
(*Local*)
VAR
	bRstErr : BOOL;
	udiRstErrOld : UDINT;
	bInitDone : BOOL;
	bInitialDone : BOOL;
	eOpsStep : eMagConvStprRunStep := MagConvStprStepNA;
	eGotoOpsStep : eMagConvStprRunStep := MagConvStprStepInit;
	eOpsStep1 : eMagConvStprRunStep := MagConvStprStepNA;
	eGotoOpsStep1 : eMagConvStprRunStep := MagConvStprStepInitDone;
	eOpsStep2 : eMagConvStprRunStep := MagConvStprStepNA;
	eGotoOpsStep2 : eMagConvStprRunStep := MagConvStprStepInit;
	fbMidChkDlyTm : TON := (PT:=T#1s);
	fbTopMidChkDlyTm : TON := (PT:=T#1s);
	udiModuleNum : UDINT;
END_VAR
```

#### Act_Alarm.st
```iecst
(** 2019-03-25 **)
ACTION Act_Alarm:

	//Error
	IF EDGEPOS(eStatus = Error) THEN

		tyAlmData.sProgNm		:= p_sProgNm;
		tyAlmData.udiCode		:= udiStatus;
		tyAlmData.eSeverity		:= AlmSeverityError;
		tyAlmData.udiRunTime	:= tyAlmData.udiRunTime + 1;
		tyAlmData.bAlm			:= TRUE;
		tyAlmData.udiModuleNum  := udiModuleNum;
		g_sOpsMagConvStpr2ProgNm		:= p_sProgNm;

		//Get Error Message
		IF tyAlmData.udiCode < 10000 OR tyAlmData.udiCode > 10099 THEN
			tyAlmData.sAlmMsg	:= 'Unknown';
			tyAlmData.sRcyMsg	:= 'Unknown';
		ELSE
			tyAlmData.sAlmMsg	:= a_tyAlmText[tyAlmData.udiCode].sAlmText;
			tyAlmData.sRcyMsg	:= a_tyAlmText[tyAlmData.udiCode].sRcyText;
		END_IF

	ELSIF bRstErr AND (tyAlmData.udiCode <> 0) THEN

		tyAlmData.udiCode		:= 0;
		tyAlmData.eSeverity		:= AlmSeverityNA;
		tyAlmData.sAlmMsg		:= '';
		tyAlmData.sRcyMsg		:= '';
		tyAlmData.bAlm			:= FALSE;
	END_IF

END_ACTION
```

#### Act_InitGlobal.st
```iecst
(** 2019-04-16 **)
ACTION Act_InitGlobal:

	(* Always Change If Project Change *)

	//Pass Data To Link
	p_bLinkOpsMnlUnloadMag ACCESS p_UIOpsMnlUnloadMag2;
	p_bLinkOpsOutMagConvStepWaitRmv ACCESS p_OpsOutMagConv2StepWaitToRmvMag;

	//Pass Data To Internal Use
	p_udiRstErr ACCESS p_RstErrReset;
	p_bRun ACCESS p_OpsRun;
	p_bStop ACCESS p_OpsStop;
	p_bStep ACCESS p_OpsStep;
//	p_sProgNm ACCESS p_NtParamOpsMagConv2StprProgNm;
	p_bNtSettingsLoadDone ACCESS p_StartupNtSettingsLoadDone;

	p_diLinkLiftBtmActualPos ACCESS p_Lifter2ActualPos;
	p_diLinkLiftBtmPos ACCESS p_McParamLifterBtmPos2;
	p_diLinkLiftTopPos ACCESS p_McParamLifterTopPos2;

	p_eStprBtmMidStat ACCESS p_PneuNoSenBtmMidStpr2Stat;
	p_eStprBtmMidStatus ACCESS p_PneuNoSenBtmMidStpr2Status;

	p_eStprBtmExitStat ACCESS p_PneuNoSenBtmExtStpr2Stat;
	p_eStprBtmExitStatus ACCESS p_PneuNoSenBtmExtStpr2Status;

	p_eStprTopEntStat ACCESS p_PneuNoSenTopEntStpr2Stat;
	p_eStprTopEntStatus ACCESS p_PneuNoSenTopEntStpr2Status;

	p_eStprTopMidStat ACCESS p_PneuNoSenTopMidStpr2Stat;
	p_eStprTopMidStatus ACCESS p_PneuNoSenTopMidStpr2Status;
	p_bStprTopMidStprExtended ACCESS p_PneuNoSenTopMidStpr2Extended;

	p_eStprTopExitStat ACCESS p_PneuNoSenTopExtStpr2Stat;
	p_eStprTopExitStatus ACCESS p_PneuNoSenTopExtStpr2Status;
	p_bStprTopExitStprExtended ACCESS p_PneuNoSenTopEntStpr2Extended;

	p_eInMagConvStatus ACCESS p_InMagConv2Status; 	//In magConv status
	p_eInMagConvStat ACCESS p_InMagConv2Stat; 		//In magConv status
	p_eOutMagConvStatus ACCESS p_OutMagConv2Status; //In magConv status
	p_eLiftMagConvStat ACCESS p_LifterMagConv2Stat; //LiftConv Status
	p_eLiftMagConvStatus ACCESS p_LifterMagConv2Status;

//	p_bBtmMagConvZ1Sen ACCESS p_DIBtmMagConvZ1Sen;
//	p_bTopMagConvZ1Sen ACCESS p_DITopMagConvZ1Sen;
	p_bBtmMagConvZ1Sen ACCESS p_DIOutMagConv2EntSen;
	p_bTopMagConvZ1Sen ACCESS p_DIInMagConv2ExtSen;

	p_bBtmMagConvMidSen ACCESS p_DIOutMagConv2MidSen; //LtoR view
	p_bTopMagConvMidSen ACCESS p_DIInMagConv2MidSen;

	p_bBtmMagConvEndSen ACCESS p_DIOutMagConv2ExtSen; //LtoR view
	p_bTopMagConvEndSen ACCESS p_DIInMagConv2EntSen;

	p_bMagPresentSen ACCESS p_DILifter2LmtSW;

	p_bEnterSig ACCESS p_OpsInMagConv2StepEntToMid;
	p_bExitSig ACCESS p_OpsOutMagConv2StepExtMag;

	(* Always Change If Project Change *)

END_ACTION
```

#### Act_InitLocal.st
```iecst
(** 2019-04-16 **)
ACTION Act_InitLocal:

	//Input Reference Link To Local Variable
	p_udiRstErr ACCESS ADR(udiRstErr);
	p_bEn ACCESS ADR(bEn);
	p_bDis ACCESS ADR(bDis);
	p_bRun ACCESS ADR(bRun);
	p_bStop ACCESS ADR(bStop);
	p_bStep ACCESS ADR(bStep);

	p_eStprBtmExitStat ACCESS ADR(eStprBtmExitStat);
	p_eStprBtmExitStatus ACCESS ADR(eStprBtmExitStatus);
	p_eStprBtmMidStat ACCESS ADR(eStprBtmMidStat);
	p_eStprBtmMidStatus ACCESS ADR(eStprBtmMidStatus);

	p_eStprTopExitStat ACCESS ADR(eStprTopExitStat);
	p_eStprTopExitStatus ACCESS ADR(eStprTopExitStatus);
	p_eStprTopMidStat ACCESS ADR(eStprTopMidStat);
	p_eStprTopMidStatus ACCESS ADR(eStprTopMidStatus);
	p_eStprTopEntStat ACCESS ADR(eStprTopEntStat);
	p_eStprTopEntStatus ACCESS ADR(eStprTopEntStatus);

	p_bLiftBtmPos ACCESS ADR(bLiftBtmPos);
	p_bLiftTopPos ACCESS ADR(bLiftTopPos);

	p_bBtmEntToLift ACCESS ADR(bBtmEntToLift);
	p_bBtmExitFromLift ACCESS ADR(bBtmExitFromLift);
	p_bTopEntToLift ACCESS ADR(bTopEntToLift);
	p_bTopExitFromLift ACCESS ADR(bTopExitFromLift);
	p_bBtmExitFromMagConv ACCESS ADR(bBtmExitFromMagConv);
	p_bTopEntFromMagConv ACCESS ADR(bTopEntFromMagConv);
	p_bBtmExitMnl ACCESS ADR(bBtmExitMnl);

	p_bBtmMagConvZ1Sen ACCESS ADR(bBtmMagConvZ1Sen);
	p_bTopMagConvZ1Sen ACCESS ADR(bTopMagConvZ1Sen);

	p_bTopMagConvMidSen ACCESS ADR(bTopMagConvMidSen);
	p_bBtmMagConvMidSen ACCESS ADR(bBtmMagConvMidSen);

	p_bBtmMagConvEndSen ACCESS ADR(bBtmMagConvEndSen);
	p_bTopMagConvEndSen ACCESS ADR(bTopMagConvEndSen);

	p_bMagPresentSen ACCESS ADR(bMagPresentSen);
	p_eLiftMagConvAct ACCESS ADR(eLiftMagConvAct);

	p_bEnterSig ACCESS ADR(bEnterSig);
	p_bExitSig ACCESS ADR(bExitSig);

	p_sProgNm ACCESS ADR(sProgNm);
	p_bNtSettingsLoadDone ACCESS ADR(bNtSettingsLoadDone);

END_ACTION
```

#### Init.st
```iecst
(** 2019-03-25 **)
PROGRAM _INIT

	(* Always Change If Project Change *)

	//Pass Address To Global Address For External Use
	//Action, State & Status

	//Alarm
	p_OpsMagConv2StprAlmData	:= ADR(tyAlmData);

	//Output
	p_OpsMagConv2StprStepTxt	:= ADR(sStepTxt);
	p_OpsMagConv2StprPaused		:= ADR(bPaused);
	p_OpsMagConv2StprBtmEntAct	:= ADR(eStprBtmEntAct);
	p_OpsMagConv2StprBtmExitAct	:= ADR(eStprBtmExitAct);
	p_OpsMagConv2StprBtmMidAct  := ADR(eStprBtmMidAct);
	p_OpsMagConv2StprTopEntAct	:= ADR(eStprTopEntAct);
	p_OpsMagConv2StprTopExitAct	:= ADR(eStprTopExitAct);
	p_OpsMagConv2StprTopMidAct	:= ADR(eStprTopMidAct);

	(* Always Change If Project Change *)

END_PROGRAM
```

#### Program Logical/Operations/MultiMag_InOutMagazineConv/OpsMagConvStpr2/Sequence

##### Act_OpsInitial.st
```iecst
(** 2019-01-16 **)
ACTION Act_OpsInitial:

	eOpsStep		:= MagConvStprStepNA;
	eGotoOpsStep	:= MagConvStprStepInit; //btm stpr
	eOpsStep1		:= MagConvStprStepNA;
	eGotoOpsStep1	:= MagConvStprStepInitDone; //top ent stpr
	eOpsStep2		:= MagConvStprStepNA;
	eGotoOpsStep2	:= MagConvStprStepInit; //top stpr

END_ACTION
```

##### Act_OpsRun.st
```iecst
(** 2019-04-16 **)
ACTION Act_OpsRun:

	IF eGotoOpsStep <> eOpsStep THEN

		CASE eGotoOpsStep OF

			ELSE
				eOpsStep	:= eGotoOpsStep;

		END_CASE

	END_IF

	IF eOpsStep = eGotoOpsStep THEN

		IF bPaused = FALSE THEN

			CASE eOpsStep OF

				MagConvStprStepInit:

					eStprBtmMidAct  := PneuActRet;
					eStprBtmExitAct	:= PneuActExt;

					IF (p_eStprBtmMidStat = PneuActRet AND p_eStprBtmMidStatus = Done) AND
						(p_eStprBtmExitStat = PneuActExt AND p_eStprBtmExitStatus = Done)
						THEN

						eStprBtmMidAct	:= PneuActIdle;
						eStprBtmExitAct	:= PneuActIdle;

						bPaused			:= p_bStop OR p_bStep;

						eGotoOpsStep	:= MagConvStprStepChkCond;

					END_IF

				MagConvStprStepChkCond:

					IF p_bBtmEntToLift THEN //opt
						eGotoOpsStep	:= MagConvStprStepBtmLiftMagEnt; //Bottom
					ELSIF p_bBtmExitFromLift THEN
						eGotoOpsStep	:= MagConvStprStepBtmLiftMagExit; //Bottom
					ELSIF p_bBtmExitFromMagConv THEN
						eGotoOpsStep    := MagConvStprStepBtmMagConvExit; //Bottom
					ELSIF p_bBtmExitMnl THEN
						eGotoOpsStep	:= MagConvStprStepBtmMagExitMnl; //Bottom
					ELSIF p_eLiftMagConvStatus = Done THEN
						eGotoOpsStep	:= MagConvStprStepDone;
					END_IF

					fbMidChkDlyTm (IN:=p_eOutMagConvStatus <> Busy);
					IF p_bBtmExitFromLift = FALSE AND p_bBtmEntToLift = FALSE AND p_bBtmExitFromMagConv = FALSE AND
						p_bBtmMagConvEndSen AND p_bBtmMagConvMidSen AND fbMidChkDlyTm.Q AND p_eInMagConvStatus <> Busy THEN
						eStprBtmMidAct  := PneuActExt;
					ELSIF fbMidChkDlyTm.Q THEN
						eStprBtmMidAct  := PneuActRet;
					END_IF

					IF ((p_eStprBtmMidStat = PneuActExt OR p_eStprBtmMidStat = PneuActRet) AND p_eStprBtmMidStatus = Done) THEN
						eStprBtmMidAct  := PneuActIdle;
						fbMidChkDlyTm (IN:=FALSE);
					END_IF

					bPaused	:= p_bStop OR p_bStep;

				MagConvStprStepBtmLiftMagEnt:

						eStprBtmMidAct  := PneuActExt;
						eStprBtmExitAct	:= PneuActRet;

					IF (p_eStprBtmMidStat = PneuActExt AND p_eStprBtmMidStatus = Done) AND
						(p_eStprBtmExitStat = PneuActRet AND p_eStprBtmExitStatus = Done) THEN

						eStprBtmMidAct  := PneuActIdle;
						eStprBtmExitAct	:= PneuActIdle;

						bPaused			:= p_bStop OR p_bStep;

						IF p_eLiftMagConvStatus = Done OR p_eLiftMagConvStatus = Idle THEN

							eGotoOpsStep	:= MagConvStprStepDone;

						END_IF

					END_IF

				MagConvStprStepBtmLiftMagExit:

					eStprBtmMidAct	:= PneuActRet;
					eStprBtmExitAct	:= PneuActExt;

					IF (p_eStprBtmMidStat = PneuActRet AND p_eStprBtmMidStatus = Done) AND
						(p_eStprBtmExitStat = PneuActExt AND p_eStprBtmExitStatus = Done) THEN

						eStprBtmMidAct   := PneuActIdle;
						eStprBtmExitAct	 := PneuActIdle;

						bPaused			:= p_bStop OR p_bStep;

						IF p_eLiftMagConvStatus = Done OR p_eLiftMagConvStatus = Idle THEN

							eGotoOpsStep	:= MagConvStprStepDone;

						END_IF
					END_IF

				MagConvStprStepBtmMagConvExit:
					eStprBtmMidAct	:= PneuActExt;
					eStprBtmExitAct	:= PneuActRet;
					IF (p_eStprBtmMidStat = PneuActExt AND p_eStprBtmMidStatus = Done) AND
						(p_eStprBtmExitStat = PneuActRet AND p_eStprBtmExitStatus = Done) THEN
						eStprBtmMidAct	:= PneuActIdle;
						eStprBtmExitAct	:= PneuActIdle;
						bPaused			:= p_bStop OR p_bStep;

						IF p_eOutMagConvStatus = Done OR p_eOutMagConvStatus = Idle THEN
							eGotoOpsStep	:= MagConvStprStepDone;
						END_IF
					END_IF

				MagConvStprStepDone:

					eStprBtmMidAct  := PneuActRet;
					eStprBtmExitAct	:= PneuActExt;

					IF (p_eStprBtmMidStat = PneuActRet AND p_eStprBtmMidStatus = Done) AND
						(p_eStprBtmExitStat = PneuActExt AND p_eStprBtmExitStatus = Done)
						THEN

						eStprBtmMidAct	:= PneuActIdle;
						eStprBtmExitAct	:= PneuActIdle;

						bPaused			:= p_bStop OR p_bStep;

						eGotoOpsStep	:= MagConvStprStepChkCond;

					END_IF
				MagConvStprStepInitDone:
					IF p_eInMagConvStatus = Done OR p_eInMagConvStatus = Idle THEN
						eStprTopEntAct  := PneuActExt;
					END_IF

					IF (p_eStprTopEntStat = PneuActExt AND p_eStprTopEntStatus = Done) THEN
						eStprTopEntAct  := PneuActIdle;
						eGotoOpsStep 	:= MagConvStprStepChkCond;
						bPaused			:= p_bStop OR p_bStep;
					END_IF

				MagConvStprStepBtmMagExitMnl:

					eStprBtmExitAct	:= PneuActRet;

					IF (p_eStprBtmExitStat = PneuActRet AND p_eStprBtmExitStatus = Done) THEN
						eStprBtmExitAct	 := PneuActIdle;

						IF p_bBtmExitMnl = FALSE THEN
							eGotoOpsStep	:= MagConvStprStepDone;
						END_IF

						bPaused			:= p_bStop OR p_bStep;
					END_IF

			END_CASE
		END_IF
	ELSE
		bPaused	:= p_bStop OR p_bStep;
	END_IF

	//==================== sequence 2 - Top entry stopper =============================================================
	IF eGotoOpsStep1 <> eOpsStep1 THEN
		CASE eGotoOpsStep1 OF
			ELSE
				eOpsStep1	:= eGotoOpsStep1;
		END_CASE
	END_IF

	IF eGotoOpsStep1 = eOpsStep1 THEN

		IF bPaused = FALSE THEN
			CASE eOpsStep1 OF
				MagConvStprStepInitDone:
					IF eOpsStep1 > MagConvStprStepInit THEN
						eStprTopEntAct  := PneuActExt;
					END_IF

					IF (p_eStprTopEntStat = PneuActExt AND p_eStprTopEntStatus = Done) THEN
						eStprTopEntAct  := PneuActIdle;
						eGotoOpsStep1 	:= MagConvStprStepChkCond;
						bPaused			:= p_bStop OR p_bStep;
					END_IF

				MagConvStprStepChkCond:
					IF p_bTopEntFromMagConv THEN
						eGotoOpsStep1    := MagConvStprStepTopMagConvEnter;
					END_IF
					bPaused	:= p_bStop OR p_bStep;

				MagConvStprStepTopMagConvEnter:
					eStprTopEntAct	:= PneuActRet;

					IF (p_eStprTopEntStat = PneuActRet AND p_eStprTopEntStatus = Done) THEN
						eStprTopEntAct   := PneuActIdle;
						eGotoOpsStep1	:= MagConvStprStepTopMagConvEnterD;
						bPaused			:= p_bStop OR p_bStep;

					END_IF
				MagConvStprStepTopMagConvEnterD:
					IF p_bTopMagConvMidSen OR (p_eInMagConvStatus <> Busy AND p_bTopMagConvEndSen =FALSE)THEN
						eStprTopEntAct	:= PneuActExt;
					END_IF

					IF (p_eStprTopEntStat = PneuActExt AND p_eStprTopEntStatus = Done) THEN
						eStprTopEntAct   := PneuActIdle;
						bPaused			:= p_bStop OR p_bStep;
						eGotoOpsStep1	:= MagConvStprStepChkCond;
					END_IF
			END_CASE
		END_IF
	ELSE
		bPaused	:= p_bStop OR p_bStep;
	END_IF

//################ sequence 3 - Top mid and ext stopper #####################################################################
	IF eGotoOpsStep2 <> eOpsStep2 THEN
		CASE eGotoOpsStep2 OF
			ELSE
				eOpsStep2	:= eGotoOpsStep2;
		END_CASE
	END_IF

	IF eGotoOpsStep2 = eOpsStep2 THEN
		IF bPaused = FALSE THEN
			CASE eOpsStep2 OF

				MagConvStprStepInit:

					eStprTopMidAct	:= PneuActRet;
					eStprTopExitAct := PneuActExt;

					IF 	(p_eStprTopMidStat = PneuActRet AND p_eStprTopMidStatus = Done) AND
						(p_eStprTopExitStat = PneuActExt AND p_eStprTopExitStatus = Done) THEN

						eStprTopMidAct	:= PneuActIdle;
						eStprTopExitAct := PneuActIdle;

						bPaused			:= p_bStop OR p_bStep;

						eGotoOpsStep2	:= MagConvStprStepChkCond;

					END_IF

				MagConvStprStepChkCond:

					IF p_bTopEntToLift THEN
						eGotoOpsStep2	:= MagConvStprStepTopLiftMagEnt;
					ELSIF p_bTopExitFromLift THEN //opt
						eGotoOpsStep2    := MagConvStprStepTopLiftMagExit;
					ELSIF p_eLiftMagConvStatus = Done THEN
						eGotoOpsStep2	:= MagConvStprStepDone;
					END_IF

					fbTopMidChkDlyTm (IN:=p_eInMagConvStatus <> Busy);
					IF p_bTopEntToLift = FALSE AND p_bTopExitFromLift = FALSE AND p_bTopEntFromMagConv = FALSE AND
						p_bTopMagConvZ1Sen AND p_bTopMagConvMidSen AND fbTopMidChkDlyTm.Q AND p_eOutMagConvStatus <> Busy THEN
						eStprTopMidAct  := PneuActExt;
					ELSIF fbTopMidChkDlyTm.Q THEN
						eStprTopMidAct  := PneuActRet;
					END_IF

					IF ((p_eStprTopMidStat = PneuActExt OR p_eStprTopMidStat = PneuActRet) AND p_eStprTopMidStatus = Done) THEN
						eStprTopMidAct  := PneuActIdle;
						fbTopMidChkDlyTm (IN:=FALSE);
					END_IF

					bPaused	:= p_bStop OR p_bStep;

				MagConvStprStepTopLiftMagEnt:
					IF p_bTopMagConvMidSen THEN
						eStprTopMidAct  := PneuActExt;
					ELSE
						eStprTopMidAct  := PneuActRet;
					END_IF
					eStprTopExitAct	:= PneuActRet;

					IF ((p_eStprTopMidStat = PneuActExt OR p_eStprTopMidStat = PneuActRet) AND p_eStprTopMidStatus = Done) AND
						(p_eStprTopExitStat = PneuActRet AND p_eStprTopExitStatus = Done) THEN

						eStprTopMidAct  := PneuActIdle;
						eStprTopExitAct	:= PneuActIdle;

						bPaused			:= p_bStop OR p_bStep;

						IF p_eLiftMagConvStatus = Done OR p_eLiftMagConvStatus = Idle THEN

							eGotoOpsStep2	:= MagConvStprStepDone;
						END_IF

					END_IF

				MagConvStprStepTopLiftMagExit:

					eStprTopMidAct	:= PneuActRet;
					eStprTopExitAct	:= PneuActRet;

					IF (p_eStprTopMidStat = PneuActRet AND p_eStprTopMidStatus = Done) AND
						(p_eStprTopExitStat = PneuActRet AND p_eStprTopExitStatus = Done) THEN

						eStprTopMidAct   := PneuActIdle;
						eStprTopExitAct	 := PneuActIdle;

						bPaused			:= p_bStop OR p_bStep;

						IF p_eLiftMagConvStatus = Done OR p_eLiftMagConvStatus = Idle THEN

							eGotoOpsStep2	:= MagConvStprStepDone;

						END_IF
					END_IF

				MagConvStprStepTopMagConvEnter:
					eStprTopEntAct	:= PneuActRet;

					IF (p_eStprTopEntStat = PneuActRet AND p_eStprTopEntStatus = Done) THEN
						eStprTopEntAct   := PneuActIdle;
						eGotoOpsStep2	:= MagConvStprStepTopMagConvEnterD;

						bPaused			:= p_bStop OR p_bStep;

					END_IF

				MagConvStprStepTopMagConvEnterD:
					IF p_bTopMagConvMidSen THEN
						eStprTopEntAct	:= PneuActExt;
					END_IF

					IF (p_eStprTopEntStat = PneuActExt AND p_eStprTopEntStatus = Done) THEN
						eStprTopEntAct   := PneuActIdle;
						bPaused			:= p_bStop OR p_bStep;
						eGotoOpsStep2	:= MagConvStprStepChkCond;
					END_IF

				MagConvStprStepDone:

					eStprTopMidAct	:= PneuActRet;
					eStprTopExitAct := PneuActExt;

					IF 	(p_eStprTopMidStat = PneuActRet AND p_eStprTopMidStatus = Done) AND
						(p_eStprTopExitStat = PneuActExt AND p_eStprTopExitStatus = Done) THEN

						eStprTopMidAct	:= PneuActIdle;
						eStprTopExitAct := PneuActIdle;

						bPaused			:= p_bStop OR p_bStep;

						eGotoOpsStep2	:= MagConvStprStepChkCond;

					END_IF

				MagConvStprStepInitDone:
					IF p_eInMagConvStatus = Done OR p_eInMagConvStatus = Idle THEN
						eStprTopEntAct  := PneuActExt;
					END_IF

					IF (p_eStprTopEntStat = PneuActExt AND p_eStprTopEntStatus = Done) THEN
						eStprTopEntAct  := PneuActIdle;
						eGotoOpsStep2 	:= MagConvStprStepChkCond;
						bPaused			:= p_bStop OR p_bStep;
					END_IF
			END_CASE
		END_IF
	ELSE
		bPaused	:= p_bStop OR p_bStep;
	END_IF

END_ACTION
```

### Program Logical/Operations/OpsPosAllwGo (IEC)

#### Init.st - Change By Project
```iecst
(** 2019-03-25 **)
PROGRAM _INIT
	p_OpsUSPosAllwGo	:= ADR(udiUSPosAllwGo);
	p_OpsDSPosAllwGo	:= ADR(udiDSPosAllwGo);
	p_OpsUSPosAllwGoStep	:= ADR(eOpsStep);
	p_OpsDSPosAllwGoStep	:= ADR(eOpsStep1);
END_PROGRAM
```

#### Act_InitGlobal.st - Change By Project
```iecst
(** 2019-04-16 **)
ACTION Act_InitGlobal:
	//Pass Data To Internal Use
	p_udiRstErr ACCESS p_RstErrReset;
	p_bRun ACCESS p_OpsRun;
	p_bStop ACCESS p_OpsStop;
	p_bStep ACCESS p_OpsStep;
	p_sProgNm ACCESS p_NtParamOpsMagConvStprProgNm;
	p_bNtSettingsLoadDone ACCESS p_StartupNtSettingsLoadDone;

	p_eUSCommMod1 ACCESS p_McParamUSCommAMod;
	p_eUSCommMod2 ACCESS p_McParamUSCommBMod;

	p_tyBufferStat1 ACCESS p_Buffer1BffrStat;
	p_tyBufferStat2 ACCESS p_Buffer2BffrStat;
	p_tyBufferStat3 ACCESS p_Buffer3BffrStat;

	p_dtBufferMagPresentTm1 ACCESS p_Buffer1MagPresentTm;
	p_dtBufferMagPresentTm2 ACCESS p_Buffer2MagPresentTm;
	p_dtBufferMagPresentTm3 ACCESS p_Buffer3MagPresentTm;

	p_bUSHermesUSRdy1 ACCESS p_USHermesAUSRdy;
	p_bUSHermesUSGdRdy1 ACCESS p_USHermesAUSGdRdy;

	p_bUSHermesUSRdy2 ACCESS p_USHermesBUSRdy;
	p_bUSHermesUSGdRdy2 ACCESS p_USHermesBUSGdRdy;

	p_bUSSMEMAUSRdy1 ACCESS p_USSMEMAAUSRdy;
	p_bUSSMEMAGdBrdRdy1 ACCESS p_USSMEMAAUSGdBrdRdy;
	p_bUSSMEMAUSRdy2 ACCESS p_USSMEMABUSRdy;
	p_bUSSMEMAGdBrdRdy2 ACCESS p_USSMEMABUSGdBrdRdy;

	p_bDSSMEMADSRdy1 ACCESS p_DSSMEMA1DSRdy;
	p_bDSSMEMADSRdy2 ACCESS p_DSSMEMA2DSRdy;
	p_bDSSMEMADSRdy3 ACCESS p_DSSMEMA3DSRdy;

	p_tyParamTravLif ACCESS p_OpsTravLifParamTravLif;
	p_bConvGdBrd ACCESS p_PshrConvGdBrd;

	p_usiLinkProdRcpCurrRcpMcMod ACCESS p_ProdRcpCurrRcp1McMod;

	p_bOpsModGoneThrough ACCESS p_OpsTravLifOpsModGonethrough;
END_ACTION
```

#### Act_Link.st - Change By Project
```iecst
(** 2018-12-11 **)
ACTION Act_Link:

	p_eULMod	:= USINT_TO_UDINT(p_usiLinkProdRcpCurrRcpMcMod);

	CASE p_eULMod OF
		ULModUnloadFrontLnA, ULModUnloadRearLnB, ULModUnloadDualLnAB:
			bBypsGdBadBrd	:= TRUE;
		ULModRejFrontLnA, ULModRejFrontLnARev, ULModRejRearLnB, ULModRejRearLnBRev, ULModRejDualLnA, ULModRejDualLnB:
			bBypsGdBadBrd	:= FALSE;
	END_CASE

	//Upstream
	IF p_eUSCommMod1 = McSetCommModHermes THEN
		bLocalUSRdy1	:= p_bUSHermesUSRdy1;
		bLocalUSGdRdy1	:= p_bUSHermesUSGdRdy1;
	ELSE
		bLocalUSRdy1	:= p_bUSSMEMAUSRdy1;
		bLocalUSGdRdy1	:= p_bUSSMEMAGdBrdRdy1;
	END_IF

	IF p_eUSCommMod2 = McSetCommModHermes THEN
		bLocalUSRdy2	:= p_bUSHermesUSRdy2;
		bLocalUSGdRdy2	:= p_bUSHermesUSGdRdy2;
	ELSE
		bLocalUSRdy2	:= p_bUSSMEMAUSRdy2;
		bLocalUSGdRdy2	:= p_bUSSMEMAGdBrdRdy2;
	END_IF

	IF p_eUSCommMod3 = McSetCommModHermes THEN
		bLocalUSRdy3	:= p_bUSHermesUSRdy3;
		bLocalUSGdRdy3	:= p_bUSHermesUSGdRdy3;
	ELSE
		bLocalUSRdy3	:= p_bUSSMEMAUSRdy3;
		bLocalUSGdRdy3	:= p_bUSSMEMAGdBrdRdy3;
	END_IF

	//Downstream
	IF p_eDSCommMod1 = McSetCommModHermes THEN
		bLocalDSRdy1	:= p_bDSHermesDSRdy1;
	ELSE
		bLocalDSRdy1	:= p_bDSSMEMADSRdy1;
	END_IF

	IF p_eDSCommMod2 = McSetCommModHermes THEN
		bLocalDSRdy2	:= p_bDSHermesDSRdy2;
	ELSE
		bLocalDSRdy2	:= p_bDSSMEMADSRdy2;
	END_IF

	IF p_eDSCommMod3 = McSetCommModHermes THEN
		bLocalDSRdy3	:= p_bDSHermesDSRdy3;
	ELSE
		bLocalDSRdy3	:= p_bDSSMEMADSRdy3;
	END_IF

END_ACTION
```

#### Act_InitLocal.st - Do Not Change!!!
```iecst
(** 2019-04-16 **)
ACTION Act_InitLocal:

	//Input Reference Link To Local Variable
	p_udiRstErr ACCESS ADR(udiRstErr);
	p_bEn ACCESS ADR(bEn);
	p_bDis ACCESS ADR(bDis);
	p_bRun ACCESS ADR(bRun);
	p_bStop ACCESS ADR(bStop);
	p_bStep ACCESS ADR(bStep);

	p_eUSCommMod1 ACCESS ADR(eUSCommMod1);
	p_eUSCommMod2 ACCESS ADR(eUSCommMod2);
	p_eUSCommMod3 ACCESS ADR(eUSCommMod3);
	p_eDSCommMod1 ACCESS ADR(eDSCommMod1);
	p_eDSCommMod2 ACCESS ADR(eDSCommMod2);
	p_eDSCommMod3 ACCESS ADR(eDSCommMod3);

	p_bUSSMEMAUSRdy3 ACCESS ADR(bUSSMEMAUSRdy3);
	p_bUSSMEMAGdBrdRdy3 ACCESS ADR(bUSSMEMAGdBrdRdy3);

	p_bDSHermesDSRdy1 ACCESS ADR(bDSHermesDSRdy1);
	p_bDSHermesDSRdy2 ACCESS ADR(bDSHermesDSRdy2);
	p_bDSHermesDSRdy3 ACCESS ADR(bDSHermesDSRdy3);

	p_sProgNm ACCESS ADR(sProgNm);
	p_bNtSettingsLoadDone ACCESS ADR(bNtSettingsLoadDone);

	p_bBypsGdBadBrd ACCESS ADR(bBypsGdBadBrd);
	p_eULMod ACCESS ADR(eULMode);

END_ACTION
```

#### Package Logical/Operations/OpsPosAllwGo/Sequence - Do Not Change!!!

#### Act_OpsInitial.st
```iecst
(** 2019-01-16 **)
ACTION Act_OpsInitial:

	eOpsStep		:= ePosUSAllwGoStepNA;
	eGotoOpsStep	:= ePosUSAllwGoStepInit;

	eOpsStep1		:= ePosDSAllwGoStepNA;
	eGotoOpsStep1	:= ePosDSAllwGoStepInit;
END_ACTION
```

#### Act_OpsRst.st
```iecst
(** 2019-03-25 **)
ACTION Act_OpsRst:

	udiUSPosAllwGo := 99;
	udiDSPosAllwGo := 99;

END_ACTION
```

#### Act_OpsRun.st
```iecst
(** 2019-04-16 **)
ACTION Act_OpsRun:
	bPaused	:= p_bStop OR p_bStep;

	IF eGotoOpsStep <> eOpsStep THEN

		CASE eGotoOpsStep OF

			ELSE
				eOpsStep	:= eGotoOpsStep;

		END_CASE

	END_IF

	IF eOpsStep = eGotoOpsStep THEN

		IF bPaused = FALSE THEN

			CASE eOpsStep OF
				ePosUSAllwGoStepInit:
					eGotoOpsStep := ePosUSAllwGoUSCheck;
//				ePosUSAllwGoStepStdBy:
//					IF p_bOpsModGoneThrough THEN
//						eGotoOpsStep := ePosUSAllwGoUSCheck;
//					END_IF

				ePosUSAllwGoUSCheck:

					a_bPosAllwSigOn[1]	:= bLocalUSRdy1;
					a_bPosAllwSigOn[2]	:= bLocalUSRdy2;
					a_bPosAllwSigOn[3]	:= bLocalUSRdy3;

					memset(ADR(a_udiPosAllwSum), 0, SIZEOF(a_udiPosAllwSum));

					FOR udi := 1 TO 3 DO
						//Priority
						a_udiPosAllwSum[udi]	:= a_udiPosAllwSum[udi] + p_tyParamTravLif.a_usiUSPriority[udi];
						//Enable
						IF p_tyParamTravLif.a_bUSDis[udi] = FALSE THEN
							a_udiPosAllwSum[udi]	:= a_udiPosAllwSum[udi] + 1000;
						END_IF
						//Signal On
						IF a_bPosAllwSigOn[udi] = TRUE THEN
							a_udiPosAllwSum[udi]	:= a_udiPosAllwSum[udi] + 2000;
						END_IF
					END_FOR

					udiUSPosAllwGo	:= 99;

					FOR udi := 1 TO 3 DO
						//Enable + Signal On
						IF a_udiPosAllwSum[udi] >= 3000 THEN

							IF udiUSPosAllwGo <> 99 THEN
								//Priority
								IF a_udiPosAllwSum[udi] < a_udiPosAllwSum[udiUSPosAllwGo] THEN
									udiUSPosAllwGo	:= udi;
								END_IF
							ELSE
								udiUSPosAllwGo	:= udi;
							END_IF
						END_IF
					END_FOR

					IF udiUSPosAllwGo = 99 THEN
						FOR udi := 1 TO 3 DO
							//Enable (Single Input)
							IF a_udiPosAllwSum[udi] >= 1000 AND a_udiPosAllwSum[udi] < 2000 THEN
								IF udiUSPosAllwGo = 99 THEN
									udiUSPosAllwGo	:= udi;
								ELSE
									udiUSPosAllwGo	:= 99;
									EXIT;
								END_IF
							END_IF
						END_FOR
					END_IF

					//eGotoOpsStep:= ePosUSAllwGoUSCheck;
			END_CASE
		END_IF
	ELSE
		bPaused	:= p_bStop OR p_bStep;
	END_IF

	IF eGotoOpsStep1 <> eOpsStep1 THEN

		CASE eGotoOpsStep1 OF

			ELSE
				eOpsStep1	:= eGotoOpsStep1;

		END_CASE

	END_IF

	IF eOpsStep1 = eGotoOpsStep1 THEN

		IF bPaused = FALSE THEN

			CASE eOpsStep1 OF
				ePosDSAllwGoStepInit:
					eGotoOpsStep1 := ePosDSAllwGoDSCheck;

//				ePosDSAllwGoStepStdBy:
//					IF p_bOpsModGoneThrough THEN
//						eGotoOpsStep := ePosUSAllwGoUSCheck;
//					END_IF

				ePosDSAllwGoDSCheck:
					a_bPosAllwSigOn[1]	:= bLocalDSRdy1;
					a_bPosAllwSigOn[2]	:= bLocalDSRdy2;
					a_bPosAllwSigOn[3]	:= bLocalDSRdy3;

					a_tyMagAllwBffrStat[1]	:= p_tyBufferStat1;
					a_tyMagAllwBffrStat[2]	:= p_tyBufferStat2;
					a_tyMagAllwBffrStat[3]	:= p_tyBufferStat3;

					IF a_bPosAllwSigOn[1] = TRUE THEN
						a_udiMagAllwMagPresentTm[1]	:= DT_TO_UDINT(p_dtBufferMagPresentTm1);
					ELSE
						a_udiMagAllwMagPresentTm[1]	:= DT_TO_UDINT(p_dtBufferMagPresentTm1)+2000000000;
					END_IF

					IF a_bPosAllwSigOn[2] = TRUE THEN
						a_udiMagAllwMagPresentTm[2]	:= DT_TO_UDINT(p_dtBufferMagPresentTm2);
					ELSE
						a_udiMagAllwMagPresentTm[2]	:= DT_TO_UDINT(p_dtBufferMagPresentTm2)+2000000000;
					END_IF

					IF a_bPosAllwSigOn[3] = TRUE THEN
						a_udiMagAllwMagPresentTm[3]	:= DT_TO_UDINT(p_dtBufferMagPresentTm3);
					ELSE
						a_udiMagAllwMagPresentTm[3]	:= DT_TO_UDINT(p_dtBufferMagPresentTm3)+2000000000;
					END_IF

					FOR udiMagPresentTm := 1 TO 3 DO
						udiCount	:= 3;

						udiCmpTm	:= a_udiMagAllwMagPresentTm[udiMagPresentTm];

						FOR udiMagPresentTm1 := 1 TO 3 DO
							IF a_udiMagAllwMagPresentTm[udiMagPresentTm1] < udiCmpTm THEN
								udiCount	:= udiCount - 1;
							END_IF
						END_FOR

						a_udiMagAllwPriority[udiMagPresentTm]	:= udiCount;
					END_FOR

					bGdChk	:= p_bConvGdBrd OR p_bBypsGdBadBrd;

					memset(ADR(a_udiPosAllwSum), 0, SIZEOF(a_udiPosAllwSum));

					FOR udi := 1 TO 3 DO
						//Priority
						//	a_udiPosAllwSum[udi]	:= a_udiPosAllwSum[udi] + p_tyParamTravLif.a_usiDSPriority[udi];
						a_udiPosAllwSum[udi]	:= a_udiPosAllwSum[udi] + a_udiMagAllwPriority[udi];
						//Enable
						IF p_tyParamTravLif.a_bDSDis[udi] = FALSE THEN
							a_udiPosAllwSum[udi]	:= a_udiPosAllwSum[udi] + 1000;
						END_IF
						//Signal On
						IF a_bPosAllwSigOn[udi] = TRUE THEN
							a_udiPosAllwSum[udi]	:= a_udiPosAllwSum[udi] + 2000;
						END_IF

						//Magazine Reject
						IF p_bBypsGdBadBrd = FALSE AND p_tyParamTravLif.a_bMagRej[udi] = TRUE THEN
							a_udiPosAllwSum[udi]	:= a_udiPosAllwSum[udi] + 6000;
						END_IF

					END_FOR

					udiDSPosAllwGo	:= 99;

					FOR udi := 1 TO 3 DO
						IF (a_udiPosAllwSum[udi] >= 3003 AND a_udiPosAllwSum[udi] < 6000 AND bGdChk = TRUE)	//Enable + Signal Allow
							OR (a_udiPosAllwSum[udi] >= 9000 AND bGdChk = FALSE) //Reject + Enable + Signal Allow
							OR (p_eULMod >= ULModUnloadDualLnAB AND (a_udiPosAllwSum[udi] >= 3000 AND a_udiPosAllwSum[udi] < 6000 AND bGdChk = TRUE))
							THEN

							IF udiDSPosAllwGo <> 99 THEN
								//Priority
								IF a_udiPosAllwSum[udi] > a_udiPosAllwSum[udiDSPosAllwGo] THEN
									udiDSPosAllwGo	:= udi;
								END_IF
							ELSE
								udiDSPosAllwGo	:= udi;
							END_IF

						END_IF

					END_FOR

					IF udiDSPosAllwGo = 99 THEN

						FOR udi := 1 TO 3 DO
							//	IF (a_udiPosAllwSum[udi] >= 1000 AND a_udiPosAllwSum[udi] < 2000 AND bGdChk = TRUE)				//Enable (Single Output)
							IF (a_udiPosAllwSum[udi] >= 3000(*3003*) AND a_udiPosAllwSum[udi] < 6000 AND bGdChk = TRUE)				//Enable (Single Output)
								//	OR (a_udiPosAllwSum[udi] >= 7000 AND a_udiPosAllwSum[udi] < 8000 AND bGdChk = FALSE) THEN	//Reject + Enable (Single Output)
								OR (a_udiPosAllwSum[udi] >= 9000 AND bGdChk = FALSE) THEN
								IF udiDSPosAllwGo = 99 THEN
									udiDSPosAllwGo	:= udi;
								ELSE
									udiDSPosAllwGo	:= 99;
									EXIT;
								END_IF

							END_IF

						END_FOR

					END_IF

			END_CASE
		END_IF
	ELSE
		bPaused	:= p_bStop OR p_bStep;
	END_IF

END_ACTION
```
